(* Logix 5000 project; controller reports 1756-L63 rev 20.11; software revision 20.04; part 26 of 52 *)

        [1809].time.Day := 15, [1809].time.Hour := 23, [1809].time.Minute := 9, [1809].time.Second := 59, [1810].log_data[0].min := 1.0, [1810].log_data[0].max := 1.0, [1810].log_data[0].total := 300.0, [1810].log_data[0].time := 300.0, [1810].log_data[0].minminute := 10, [1810].log_data[0].maxminute := 10, [1810].log_data[0].valid := 1, [1810].log_data[1].valid := 1, [1810].log_data[2].valid := 1, [1810].log_data[3].valid := 1, [1810].log_data[4].valid := 1, [1810].log_data[5].valid := 1, [1810].log_data[6].valid := 1, [1810].log_data[7].valid := 1, [1810].log_data[8].valid := 1, [1810].log_data[9].valid := 1, [1810].log_data[10].valid := 1, [1810].log_data[11].valid := 1, [1810].log_data[12].valid := 1, [1810].log_data[13].valid := 1, [1810].log_data[14].valid := 1, [1810].log_data[15].valid := 1, [1810].log_data[16].valid := 1, [1810].log_data[17].valid := 1, [1810].log_data[18].valid := 1, [1810].log_data[19].valid := 1, [1810].time.Year := 2023, [1810].time.Month := 1, [1810].time.Day := 15, [1810].time.Hour := 23, [1810].time.Minute := 14, [1810].time.Second := 59, [1811].log_data[0].min := 1.0, [1811].log_data[0].max := 1.0, [1811].log_data[0].total := 300.0, [1811].log_data[0].time := 300.0, [1811].log_data[0].minminute := 15, [1811].log_data[0].maxminute := 15, [1811].log_data[0].valid := 1, [1811].log_data[1].valid := 1, [1811].log_data[2].valid := 1, [1811].log_data[3].valid := 1, [1811].log_data[4].valid := 1, [1811].log_data[5].valid := 1, [1811].log_data[6].valid := 1, [1811].log_data[7].valid := 1, [1811].log_data[8].valid := 1, [1811].log_data[9].valid := 1, [1811].log_data[10].valid := 1, [1811].log_data[11].valid := 1, [1811].log_data[12].valid := 1, [1811].log_data[13].valid := 1, [1811].log_data[14].valid := 1, [1811].log_data[15].valid := 1, [1811].log_data[16].valid := 1, [1811].log_data[17].valid := 1,
        [1811].log_data[18].valid := 1, [1811].log_data[19].valid := 1, [1811].time.Year := 2023, [1811].time.Month := 1, [1811].time.Day := 15, [1811].time.Hour := 23, [1811].time.Minute := 19, [1811].time.Second := 59, [1812].log_data[0].min := 1.0, [1812].log_data[0].max := 1.0, [1812].log_data[0].total := 300.0, [1812].log_data[0].time := 300.0, [1812].log_data[0].minminute := 20, [1812].log_data[0].maxminute := 20, [1812].log_data[0].valid := 1, [1812].log_data[1].valid := 1, [1812].log_data[2].valid := 1, [1812].log_data[3].valid := 1, [1812].log_data[4].valid := 1, [1812].log_data[5].valid := 1, [1812].log_data[6].valid := 1, [1812].log_data[7].valid := 1, [1812].log_data[8].valid := 1, [1812].log_data[9].valid := 1, [1812].log_data[10].valid := 1, [1812].log_data[11].valid := 1, [1812].log_data[12].valid := 1, [1812].log_data[13].valid := 1, [1812].log_data[14].valid := 1, [1812].log_data[15].valid := 1, [1812].log_data[16].valid := 1, [1812].log_data[17].valid := 1, [1812].log_data[18].valid := 1, [1812].log_data[19].valid := 1, [1812].time.Year := 2023, [1812].time.Month := 1, [1812].time.Day := 15, [1812].time.Hour := 23, [1812].time.Minute := 24, [1812].time.Second := 59, [1813].log_data[0].min := 1.0, [1813].log_data[0].max := 1.0, [1813].log_data[0].total := 300.0, [1813].log_data[0].time := 300.0, [1813].log_data[0].minminute := 25, [1813].log_data[0].maxminute := 25, [1813].log_data[0].valid := 1, [1813].log_data[1].valid := 1, [1813].log_data[2].valid := 1, [1813].log_data[3].valid := 1, [1813].log_data[4].valid := 1, [1813].log_data[5].valid := 1, [1813].log_data[6].valid := 1, [1813].log_data[7].valid := 1, [1813].log_data[8].valid := 1, [1813].log_data[9].valid := 1, [1813].log_data[10].valid := 1, [1813].log_data[11].valid := 1, [1813].log_data[12].valid := 1, [1813].log_data[13].valid := 1,
        [1813].log_data[14].valid := 1, [1813].log_data[15].valid := 1, [1813].log_data[16].valid := 1, [1813].log_data[17].valid := 1, [1813].log_data[18].valid := 1, [1813].log_data[19].valid := 1, [1813].time.Year := 2023, [1813].time.Month := 1, [1813].time.Day := 15, [1813].time.Hour := 23, [1813].time.Minute := 29, [1813].time.Second := 59, [1814].log_data[0].min := 1.0, [1814].log_data[0].max := 1.0, [1814].log_data[0].total := 300.0, [1814].log_data[0].time := 300.0, [1814].log_data[0].minminute := 30, [1814].log_data[0].maxminute := 30, [1814].log_data[0].valid := 1, [1814].log_data[1].valid := 1, [1814].log_data[2].valid := 1, [1814].log_data[3].valid := 1, [1814].log_data[4].valid := 1, [1814].log_data[5].valid := 1, [1814].log_data[6].valid := 1, [1814].log_data[7].valid := 1, [1814].log_data[8].valid := 1, [1814].log_data[9].valid := 1, [1814].log_data[10].valid := 1, [1814].log_data[11].valid := 1, [1814].log_data[12].valid := 1, [1814].log_data[13].valid := 1, [1814].log_data[14].valid := 1, [1814].log_data[15].valid := 1, [1814].log_data[16].valid := 1, [1814].log_data[17].valid := 1, [1814].log_data[18].valid := 1, [1814].log_data[19].valid := 1, [1814].time.Year := 2023, [1814].time.Month := 1, [1814].time.Day := 15, [1814].time.Hour := 23, [1814].time.Minute := 34, [1814].time.Second := 59, [1815].log_data[0].min := 1.0, [1815].log_data[0].max := 1.0, [1815].log_data[0].total := 300.0, [1815].log_data[0].time := 300.0, [1815].log_data[0].minminute := 35, [1815].log_data[0].maxminute := 35, [1815].log_data[0].valid := 1, [1815].log_data[1].valid := 1, [1815].log_data[2].valid := 1, [1815].log_data[3].valid := 1, [1815].log_data[4].valid := 1, [1815].log_data[5].valid := 1, [1815].log_data[6].valid := 1, [1815].log_data[7].valid := 1, [1815].log_data[8].valid := 1, [1815].log_data[9].valid := 1,
        [1815].log_data[10].valid := 1, [1815].log_data[11].valid := 1, [1815].log_data[12].valid := 1, [1815].log_data[13].valid := 1, [1815].log_data[14].valid := 1, [1815].log_data[15].valid := 1, [1815].log_data[16].valid := 1, [1815].log_data[17].valid := 1, [1815].log_data[18].valid := 1, [1815].log_data[19].valid := 1, [1815].time.Year := 2023, [1815].time.Month := 1, [1815].time.Day := 15, [1815].time.Hour := 23, [1815].time.Minute := 39, [1815].time.Second := 59, [1816].log_data[0].min := 1.0, [1816].log_data[0].max := 1.0, [1816].log_data[0].total := 300.0, [1816].log_data[0].time := 300.0, [1816].log_data[0].minminute := 40, [1816].log_data[0].maxminute := 40, [1816].log_data[0].valid := 1, [1816].log_data[1].valid := 1, [1816].log_data[2].valid := 1, [1816].log_data[3].valid := 1, [1816].log_data[4].valid := 1, [1816].log_data[5].valid := 1, [1816].log_data[6].valid := 1, [1816].log_data[7].valid := 1, [1816].log_data[8].valid := 1, [1816].log_data[9].valid := 1, [1816].log_data[10].valid := 1, [1816].log_data[11].valid := 1, [1816].log_data[12].valid := 1, [1816].log_data[13].valid := 1, [1816].log_data[14].valid := 1, [1816].log_data[15].valid := 1, [1816].log_data[16].valid := 1, [1816].log_data[17].valid := 1, [1816].log_data[18].valid := 1, [1816].log_data[19].valid := 1, [1816].time.Year := 2023, [1816].time.Month := 1, [1816].time.Day := 15, [1816].time.Hour := 23, [1816].time.Minute := 44, [1816].time.Second := 59, [1817].log_data[0].min := 1.0, [1817].log_data[0].max := 1.0, [1817].log_data[0].total := 300.0, [1817].log_data[0].time := 300.0, [1817].log_data[0].minminute := 45, [1817].log_data[0].maxminute := 45, [1817].log_data[0].valid := 1, [1817].log_data[1].valid := 1, [1817].log_data[2].valid := 1, [1817].log_data[3].valid := 1, [1817].log_data[4].valid := 1, [1817].log_data[5].valid := 1,
        [1817].log_data[6].valid := 1, [1817].log_data[7].valid := 1, [1817].log_data[8].valid := 1, [1817].log_data[9].valid := 1, [1817].log_data[10].valid := 1, [1817].log_data[11].valid := 1, [1817].log_data[12].valid := 1, [1817].log_data[13].valid := 1, [1817].log_data[14].valid := 1, [1817].log_data[15].valid := 1, [1817].log_data[16].valid := 1, [1817].log_data[17].valid := 1, [1817].log_data[18].valid := 1, [1817].log_data[19].valid := 1, [1817].time.Year := 2023, [1817].time.Month := 1, [1817].time.Day := 15, [1817].time.Hour := 23, [1817].time.Minute := 49, [1817].time.Second := 59, [1818].log_data[0].min := 1.0, [1818].log_data[0].max := 1.0, [1818].log_data[0].total := 300.0, [1818].log_data[0].time := 300.0, [1818].log_data[0].minminute := 50, [1818].log_data[0].maxminute := 50, [1818].log_data[0].valid := 1, [1818].log_data[1].valid := 1, [1818].log_data[2].valid := 1, [1818].log_data[3].valid := 1, [1818].log_data[4].valid := 1, [1818].log_data[5].valid := 1, [1818].log_data[6].valid := 1, [1818].log_data[7].valid := 1, [1818].log_data[8].valid := 1, [1818].log_data[9].valid := 1, [1818].log_data[10].valid := 1, [1818].log_data[11].valid := 1, [1818].log_data[12].valid := 1, [1818].log_data[13].valid := 1, [1818].log_data[14].valid := 1, [1818].log_data[15].valid := 1, [1818].log_data[16].valid := 1, [1818].log_data[17].valid := 1, [1818].log_data[18].valid := 1, [1818].log_data[19].valid := 1, [1818].time.Year := 2023, [1818].time.Month := 1, [1818].time.Day := 15, [1818].time.Hour := 23, [1818].time.Minute := 54, [1818].time.Second := 59, [1819].log_data[0].min := 1.0, [1819].log_data[0].max := 1.0, [1819].log_data[0].total := 300.0, [1819].log_data[0].time := 300.0, [1819].log_data[0].minminute := 55, [1819].log_data[0].maxminute := 55, [1819].log_data[0].valid := 1, [1819].log_data[1].valid := 1,
        [1819].log_data[2].valid := 1, [1819].log_data[3].valid := 1, [1819].log_data[4].valid := 1, [1819].log_data[5].valid := 1, [1819].log_data[6].valid := 1, [1819].log_data[7].valid := 1, [1819].log_data[8].valid := 1, [1819].log_data[9].valid := 1, [1819].log_data[10].valid := 1, [1819].log_data[11].valid := 1, [1819].log_data[12].valid := 1, [1819].log_data[13].valid := 1, [1819].log_data[14].valid := 1, [1819].log_data[15].valid := 1, [1819].log_data[16].valid := 1, [1819].log_data[17].valid := 1, [1819].log_data[18].valid := 1, [1819].log_data[19].valid := 1, [1819].time.Year := 2023, [1819].time.Month := 1, [1819].time.Day := 15, [1819].time.Hour := 23, [1819].time.Minute := 59, [1819].time.Second := 59, [1820].log_data[0].min := 1.0, [1820].log_data[0].max := 1.0, [1820].log_data[0].total := 300.0, [1820].log_data[0].time := 300.0, [1820].log_data[0].valid := 1, [1820].log_data[1].valid := 1, [1820].log_data[2].valid := 1, [1820].log_data[3].valid := 1, [1820].log_data[4].valid := 1, [1820].log_data[5].valid := 1, [1820].log_data[6].valid := 1, [1820].log_data[7].valid := 1, [1820].log_data[8].valid := 1, [1820].log_data[9].valid := 1, [1820].log_data[10].valid := 1, [1820].log_data[11].valid := 1, [1820].log_data[12].valid := 1, [1820].log_data[13].valid := 1, [1820].log_data[14].valid := 1, [1820].log_data[15].valid := 1, [1820].log_data[16].valid := 1, [1820].log_data[17].valid := 1, [1820].log_data[18].valid := 1, [1820].log_data[19].valid := 1, [1820].time.Year := 2023, [1820].time.Month := 1, [1820].time.Day := 16, [1820].time.Minute := 4, [1820].time.Second := 59, [1821].log_data[0].min := 1.0, [1821].log_data[0].max := 1.0, [1821].log_data[0].total := 300.0, [1821].log_data[0].time := 300.0, [1821].log_data[0].minminute := 5, [1821].log_data[0].maxminute := 5, [1821].log_data[0].valid := 1,
        [1821].log_data[1].valid := 1, [1821].log_data[2].valid := 1, [1821].log_data[3].valid := 1, [1821].log_data[4].valid := 1, [1821].log_data[5].valid := 1, [1821].log_data[6].valid := 1, [1821].log_data[7].valid := 1, [1821].log_data[8].valid := 1, [1821].log_data[9].valid := 1, [1821].log_data[10].valid := 1, [1821].log_data[11].valid := 1, [1821].log_data[12].valid := 1, [1821].log_data[13].valid := 1, [1821].log_data[14].valid := 1, [1821].log_data[15].valid := 1, [1821].log_data[16].valid := 1, [1821].log_data[17].valid := 1, [1821].log_data[18].valid := 1, [1821].log_data[19].valid := 1, [1821].time.Year := 2023, [1821].time.Month := 1, [1821].time.Day := 16, [1821].time.Minute := 9, [1821].time.Second := 59, [1822].log_data[0].min := 1.0, [1822].log_data[0].max := 1.0, [1822].log_data[0].total := 300.0, [1822].log_data[0].time := 300.0, [1822].log_data[0].minminute := 10, [1822].log_data[0].maxminute := 10, [1822].log_data[0].valid := 1, [1822].log_data[1].valid := 1, [1822].log_data[2].valid := 1, [1822].log_data[3].valid := 1, [1822].log_data[4].valid := 1, [1822].log_data[5].valid := 1, [1822].log_data[6].valid := 1, [1822].log_data[7].valid := 1, [1822].log_data[8].valid := 1, [1822].log_data[9].valid := 1, [1822].log_data[10].valid := 1, [1822].log_data[11].valid := 1, [1822].log_data[12].valid := 1, [1822].log_data[13].valid := 1, [1822].log_data[14].valid := 1, [1822].log_data[15].valid := 1, [1822].log_data[16].valid := 1, [1822].log_data[17].valid := 1, [1822].log_data[18].valid := 1, [1822].log_data[19].valid := 1, [1822].time.Year := 2023, [1822].time.Month := 1, [1822].time.Day := 16, [1822].time.Minute := 14, [1822].time.Second := 59, [1823].log_data[0].min := 1.0, [1823].log_data[0].max := 1.0, [1823].log_data[0].total := 300.0, [1823].log_data[0].time := 300.0, [1823].log_data[0].minminute := 15,
        [1823].log_data[0].maxminute := 15, [1823].log_data[0].valid := 1, [1823].log_data[1].valid := 1, [1823].log_data[2].valid := 1, [1823].log_data[3].valid := 1, [1823].log_data[4].valid := 1, [1823].log_data[5].valid := 1, [1823].log_data[6].valid := 1, [1823].log_data[7].valid := 1, [1823].log_data[8].valid := 1, [1823].log_data[9].valid := 1, [1823].log_data[10].valid := 1, [1823].log_data[11].valid := 1, [1823].log_data[12].valid := 1, [1823].log_data[13].valid := 1, [1823].log_data[14].valid := 1, [1823].log_data[15].valid := 1, [1823].log_data[16].valid := 1, [1823].log_data[17].valid := 1, [1823].log_data[18].valid := 1, [1823].log_data[19].valid := 1, [1823].time.Year := 2023, [1823].time.Month := 1, [1823].time.Day := 16, [1823].time.Minute := 19, [1823].time.Second := 59, [1824].log_data[0].min := 1.0, [1824].log_data[0].max := 1.0, [1824].log_data[0].total := 300.0, [1824].log_data[0].time := 300.0, [1824].log_data[0].minminute := 20, [1824].log_data[0].maxminute := 20, [1824].log_data[0].valid := 1, [1824].log_data[1].valid := 1, [1824].log_data[2].valid := 1, [1824].log_data[3].valid := 1, [1824].log_data[4].valid := 1, [1824].log_data[5].valid := 1, [1824].log_data[6].valid := 1, [1824].log_data[7].valid := 1, [1824].log_data[8].valid := 1, [1824].log_data[9].valid := 1, [1824].log_data[10].valid := 1, [1824].log_data[11].valid := 1, [1824].log_data[12].valid := 1, [1824].log_data[13].valid := 1, [1824].log_data[14].valid := 1, [1824].log_data[15].valid := 1, [1824].log_data[16].valid := 1, [1824].log_data[17].valid := 1, [1824].log_data[18].valid := 1, [1824].log_data[19].valid := 1, [1824].time.Year := 2023, [1824].time.Month := 1, [1824].time.Day := 16, [1824].time.Minute := 24, [1824].time.Second := 59, [1825].log_data[0].min := 1.0, [1825].log_data[0].max := 1.0, [1825].log_data[0].total := 300.0,
        [1825].log_data[0].time := 300.0, [1825].log_data[0].minminute := 25, [1825].log_data[0].maxminute := 25, [1825].log_data[0].valid := 1, [1825].log_data[1].valid := 1, [1825].log_data[2].valid := 1, [1825].log_data[3].valid := 1, [1825].log_data[4].valid := 1, [1825].log_data[5].valid := 1, [1825].log_data[6].valid := 1, [1825].log_data[7].valid := 1, [1825].log_data[8].valid := 1, [1825].log_data[9].valid := 1, [1825].log_data[10].valid := 1, [1825].log_data[11].valid := 1, [1825].log_data[12].valid := 1, [1825].log_data[13].valid := 1, [1825].log_data[14].valid := 1, [1825].log_data[15].valid := 1, [1825].log_data[16].valid := 1, [1825].log_data[17].valid := 1, [1825].log_data[18].valid := 1, [1825].log_data[19].valid := 1, [1825].time.Year := 2023, [1825].time.Month := 1, [1825].time.Day := 16, [1825].time.Minute := 29, [1825].time.Second := 59, [1826].log_data[0].min := 1.0, [1826].log_data[0].max := 1.0, [1826].log_data[0].total := 300.0, [1826].log_data[0].time := 300.0, [1826].log_data[0].minminute := 30, [1826].log_data[0].maxminute := 30, [1826].log_data[0].valid := 1, [1826].log_data[1].valid := 1, [1826].log_data[2].valid := 1, [1826].log_data[3].valid := 1, [1826].log_data[4].valid := 1, [1826].log_data[5].valid := 1, [1826].log_data[6].valid := 1, [1826].log_data[7].valid := 1, [1826].log_data[8].valid := 1, [1826].log_data[9].valid := 1, [1826].log_data[10].valid := 1, [1826].log_data[11].valid := 1, [1826].log_data[12].valid := 1, [1826].log_data[13].valid := 1, [1826].log_data[14].valid := 1, [1826].log_data[15].valid := 1, [1826].log_data[16].valid := 1, [1826].log_data[17].valid := 1, [1826].log_data[18].valid := 1, [1826].log_data[19].valid := 1, [1826].time.Year := 2023, [1826].time.Month := 1, [1826].time.Day := 16, [1826].time.Minute := 34, [1826].time.Second := 59, [1827].log_data[0].min := 1.0,
        [1827].log_data[0].max := 1.0, [1827].log_data[0].total := 300.0, [1827].log_data[0].time := 300.0, [1827].log_data[0].minminute := 35, [1827].log_data[0].maxminute := 35, [1827].log_data[0].valid := 1, [1827].log_data[1].valid := 1, [1827].log_data[2].valid := 1, [1827].log_data[3].valid := 1, [1827].log_data[4].valid := 1, [1827].log_data[5].valid := 1, [1827].log_data[6].valid := 1, [1827].log_data[7].valid := 1, [1827].log_data[8].valid := 1, [1827].log_data[9].valid := 1, [1827].log_data[10].valid := 1, [1827].log_data[11].valid := 1, [1827].log_data[12].valid := 1, [1827].log_data[13].valid := 1, [1827].log_data[14].valid := 1, [1827].log_data[15].valid := 1, [1827].log_data[16].valid := 1, [1827].log_data[17].valid := 1, [1827].log_data[18].valid := 1, [1827].log_data[19].valid := 1, [1827].time.Year := 2023, [1827].time.Month := 1, [1827].time.Day := 16, [1827].time.Minute := 39, [1827].time.Second := 59, [1828].log_data[0].min := 1.0, [1828].log_data[0].max := 1.0, [1828].log_data[0].total := 300.0, [1828].log_data[0].time := 300.0, [1828].log_data[0].minminute := 40, [1828].log_data[0].maxminute := 40, [1828].log_data[0].valid := 1, [1828].log_data[1].valid := 1, [1828].log_data[2].valid := 1, [1828].log_data[3].valid := 1, [1828].log_data[4].valid := 1, [1828].log_data[5].valid := 1, [1828].log_data[6].valid := 1, [1828].log_data[7].valid := 1, [1828].log_data[8].valid := 1, [1828].log_data[9].valid := 1, [1828].log_data[10].valid := 1, [1828].log_data[11].valid := 1, [1828].log_data[12].valid := 1, [1828].log_data[13].valid := 1, [1828].log_data[14].valid := 1, [1828].log_data[15].valid := 1, [1828].log_data[16].valid := 1, [1828].log_data[17].valid := 1, [1828].log_data[18].valid := 1, [1828].log_data[19].valid := 1, [1828].time.Year := 2023, [1828].time.Month := 1, [1828].time.Day := 16, [1828].time.Minute := 44,
        [1828].time.Second := 59, [1829].log_data[0].min := 1.0, [1829].log_data[0].max := 1.0, [1829].log_data[0].total := 300.0, [1829].log_data[0].time := 300.0, [1829].log_data[0].minminute := 45, [1829].log_data[0].maxminute := 45, [1829].log_data[0].valid := 1, [1829].log_data[1].valid := 1, [1829].log_data[2].valid := 1, [1829].log_data[3].valid := 1, [1829].log_data[4].valid := 1, [1829].log_data[5].valid := 1, [1829].log_data[6].valid := 1, [1829].log_data[7].valid := 1, [1829].log_data[8].valid := 1, [1829].log_data[9].valid := 1, [1829].log_data[10].valid := 1, [1829].log_data[11].valid := 1, [1829].log_data[12].valid := 1, [1829].log_data[13].valid := 1, [1829].log_data[14].valid := 1, [1829].log_data[15].valid := 1, [1829].log_data[16].valid := 1, [1829].log_data[17].valid := 1, [1829].log_data[18].valid := 1, [1829].log_data[19].valid := 1, [1829].time.Year := 2023, [1829].time.Month := 1, [1829].time.Day := 16, [1829].time.Minute := 49, [1829].time.Second := 59, [1830].log_data[0].min := 1.0, [1830].log_data[0].max := 1.0, [1830].log_data[0].total := 300.0, [1830].log_data[0].time := 300.0, [1830].log_data[0].minminute := 50, [1830].log_data[0].maxminute := 50, [1830].log_data[0].valid := 1, [1830].log_data[1].valid := 1, [1830].log_data[2].valid := 1, [1830].log_data[3].valid := 1, [1830].log_data[4].valid := 1, [1830].log_data[5].valid := 1, [1830].log_data[6].valid := 1, [1830].log_data[7].valid := 1, [1830].log_data[8].valid := 1, [1830].log_data[9].valid := 1, [1830].log_data[10].valid := 1, [1830].log_data[11].valid := 1, [1830].log_data[12].valid := 1, [1830].log_data[13].valid := 1, [1830].log_data[14].valid := 1, [1830].log_data[15].valid := 1, [1830].log_data[16].valid := 1, [1830].log_data[17].valid := 1, [1830].log_data[18].valid := 1, [1830].log_data[19].valid := 1, [1830].time.Year := 2023, [1830].time.Month := 1,
        [1830].time.Day := 16, [1830].time.Minute := 54, [1830].time.Second := 59, [1831].log_data[0].min := 1.0, [1831].log_data[0].max := 1.0, [1831].log_data[0].total := 300.0, [1831].log_data[0].time := 300.0, [1831].log_data[0].minminute := 55, [1831].log_data[0].maxminute := 55, [1831].log_data[0].valid := 1, [1831].log_data[1].valid := 1, [1831].log_data[2].valid := 1, [1831].log_data[3].valid := 1, [1831].log_data[4].valid := 1, [1831].log_data[5].valid := 1, [1831].log_data[6].valid := 1, [1831].log_data[7].valid := 1, [1831].log_data[8].valid := 1, [1831].log_data[9].valid := 1, [1831].log_data[10].valid := 1, [1831].log_data[11].valid := 1, [1831].log_data[12].valid := 1, [1831].log_data[13].valid := 1, [1831].log_data[14].valid := 1, [1831].log_data[15].valid := 1, [1831].log_data[16].valid := 1, [1831].log_data[17].valid := 1, [1831].log_data[18].valid := 1, [1831].log_data[19].valid := 1, [1831].time.Year := 2023, [1831].time.Month := 1, [1831].time.Day := 16, [1831].time.Minute := 59, [1831].time.Second := 59, [1832].log_data[0].min := 1.0, [1832].log_data[0].max := 1.0, [1832].log_data[0].total := 300.0, [1832].log_data[0].time := 300.0, [1832].log_data[0].valid := 1, [1832].log_data[1].valid := 1, [1832].log_data[2].valid := 1, [1832].log_data[3].valid := 1, [1832].log_data[4].valid := 1, [1832].log_data[5].valid := 1, [1832].log_data[6].valid := 1, [1832].log_data[7].valid := 1, [1832].log_data[8].valid := 1, [1832].log_data[9].valid := 1, [1832].log_data[10].valid := 1, [1832].log_data[11].valid := 1, [1832].log_data[12].valid := 1, [1832].log_data[13].valid := 1, [1832].log_data[14].valid := 1, [1832].log_data[15].valid := 1, [1832].log_data[16].valid := 1, [1832].log_data[17].valid := 1, [1832].log_data[18].valid := 1, [1832].log_data[19].valid := 1, [1832].time.Year := 2023, [1832].time.Month := 1,
        [1832].time.Day := 16, [1832].time.Hour := 1, [1832].time.Minute := 4, [1832].time.Second := 59, [1833].log_data[0].min := 1.0, [1833].log_data[0].max := 1.0, [1833].log_data[0].total := 300.0, [1833].log_data[0].time := 300.0, [1833].log_data[0].minminute := 5, [1833].log_data[0].maxminute := 5, [1833].log_data[0].valid := 1, [1833].log_data[1].valid := 1, [1833].log_data[2].valid := 1, [1833].log_data[3].valid := 1, [1833].log_data[4].valid := 1, [1833].log_data[5].valid := 1, [1833].log_data[6].valid := 1, [1833].log_data[7].valid := 1, [1833].log_data[8].valid := 1, [1833].log_data[9].valid := 1, [1833].log_data[10].valid := 1, [1833].log_data[11].valid := 1, [1833].log_data[12].valid := 1, [1833].log_data[13].valid := 1, [1833].log_data[14].valid := 1, [1833].log_data[15].valid := 1, [1833].log_data[16].valid := 1, [1833].log_data[17].valid := 1, [1833].log_data[18].valid := 1, [1833].log_data[19].valid := 1, [1833].time.Year := 2023, [1833].time.Month := 1, [1833].time.Day := 16, [1833].time.Hour := 1, [1833].time.Minute := 9, [1833].time.Second := 59, [1834].log_data[0].min := 1.0, [1834].log_data[0].max := 1.0, [1834].log_data[0].total := 300.0, [1834].log_data[0].time := 300.0, [1834].log_data[0].minminute := 10, [1834].log_data[0].maxminute := 10, [1834].log_data[0].valid := 1, [1834].log_data[1].valid := 1, [1834].log_data[2].valid := 1, [1834].log_data[3].valid := 1, [1834].log_data[4].valid := 1, [1834].log_data[5].valid := 1, [1834].log_data[6].valid := 1, [1834].log_data[7].valid := 1, [1834].log_data[8].valid := 1, [1834].log_data[9].valid := 1, [1834].log_data[10].valid := 1, [1834].log_data[11].valid := 1, [1834].log_data[12].valid := 1, [1834].log_data[13].valid := 1, [1834].log_data[14].valid := 1, [1834].log_data[15].valid := 1, [1834].log_data[16].valid := 1, [1834].log_data[17].valid := 1,
        [1834].log_data[18].valid := 1, [1834].log_data[19].valid := 1, [1834].time.Year := 2023, [1834].time.Month := 1, [1834].time.Day := 16, [1834].time.Hour := 1, [1834].time.Minute := 14, [1834].time.Second := 59, [1835].log_data[0].min := 1.0, [1835].log_data[0].max := 1.0, [1835].log_data[0].total := 300.0, [1835].log_data[0].time := 300.0, [1835].log_data[0].minminute := 15, [1835].log_data[0].maxminute := 15, [1835].log_data[0].valid := 1, [1835].log_data[1].valid := 1, [1835].log_data[2].valid := 1, [1835].log_data[3].valid := 1, [1835].log_data[4].valid := 1, [1835].log_data[5].valid := 1, [1835].log_data[6].valid := 1, [1835].log_data[7].valid := 1, [1835].log_data[8].valid := 1, [1835].log_data[9].valid := 1, [1835].log_data[10].valid := 1, [1835].log_data[11].valid := 1, [1835].log_data[12].valid := 1, [1835].log_data[13].valid := 1, [1835].log_data[14].valid := 1, [1835].log_data[15].valid := 1, [1835].log_data[16].valid := 1, [1835].log_data[17].valid := 1, [1835].log_data[18].valid := 1, [1835].log_data[19].valid := 1, [1835].time.Year := 2023, [1835].time.Month := 1, [1835].time.Day := 16, [1835].time.Hour := 1, [1835].time.Minute := 19, [1835].time.Second := 59, [1836].log_data[0].min := 1.0, [1836].log_data[0].max := 1.0, [1836].log_data[0].total := 300.0, [1836].log_data[0].time := 300.0, [1836].log_data[0].minminute := 20, [1836].log_data[0].maxminute := 20, [1836].log_data[0].valid := 1, [1836].log_data[1].valid := 1, [1836].log_data[2].valid := 1, [1836].log_data[3].valid := 1, [1836].log_data[4].valid := 1, [1836].log_data[5].valid := 1, [1836].log_data[6].valid := 1, [1836].log_data[7].valid := 1, [1836].log_data[8].valid := 1, [1836].log_data[9].valid := 1, [1836].log_data[10].valid := 1, [1836].log_data[11].valid := 1, [1836].log_data[12].valid := 1, [1836].log_data[13].valid := 1,
        [1836].log_data[14].valid := 1, [1836].log_data[15].valid := 1, [1836].log_data[16].valid := 1, [1836].log_data[17].valid := 1, [1836].log_data[18].valid := 1, [1836].log_data[19].valid := 1, [1836].time.Year := 2023, [1836].time.Month := 1, [1836].time.Day := 16, [1836].time.Hour := 1, [1836].time.Minute := 24, [1836].time.Second := 59, [1837].log_data[0].min := 1.0, [1837].log_data[0].max := 1.0, [1837].log_data[0].total := 300.0, [1837].log_data[0].time := 300.0, [1837].log_data[0].minminute := 25, [1837].log_data[0].maxminute := 25, [1837].log_data[0].valid := 1, [1837].log_data[1].valid := 1, [1837].log_data[2].valid := 1, [1837].log_data[3].valid := 1, [1837].log_data[4].valid := 1, [1837].log_data[5].valid := 1, [1837].log_data[6].valid := 1, [1837].log_data[7].valid := 1, [1837].log_data[8].valid := 1, [1837].log_data[9].valid := 1, [1837].log_data[10].valid := 1, [1837].log_data[11].valid := 1, [1837].log_data[12].valid := 1, [1837].log_data[13].valid := 1, [1837].log_data[14].valid := 1, [1837].log_data[15].valid := 1, [1837].log_data[16].valid := 1, [1837].log_data[17].valid := 1, [1837].log_data[18].valid := 1, [1837].log_data[19].valid := 1, [1837].time.Year := 2023, [1837].time.Month := 1, [1837].time.Day := 16, [1837].time.Hour := 1, [1837].time.Minute := 29, [1837].time.Second := 59, [1838].log_data[0].min := 1.0, [1838].log_data[0].max := 1.0, [1838].log_data[0].total := 300.0, [1838].log_data[0].time := 300.0, [1838].log_data[0].minminute := 30, [1838].log_data[0].maxminute := 30, [1838].log_data[0].valid := 1, [1838].log_data[1].valid := 1, [1838].log_data[2].valid := 1, [1838].log_data[3].valid := 1, [1838].log_data[4].valid := 1, [1838].log_data[5].valid := 1, [1838].log_data[6].valid := 1, [1838].log_data[7].valid := 1, [1838].log_data[8].valid := 1, [1838].log_data[9].valid := 1,
        [1838].log_data[10].valid := 1, [1838].log_data[11].valid := 1, [1838].log_data[12].valid := 1, [1838].log_data[13].valid := 1, [1838].log_data[14].valid := 1, [1838].log_data[15].valid := 1, [1838].log_data[16].valid := 1, [1838].log_data[17].valid := 1, [1838].log_data[18].valid := 1, [1838].log_data[19].valid := 1, [1838].time.Year := 2023, [1838].time.Month := 1, [1838].time.Day := 16, [1838].time.Hour := 1, [1838].time.Minute := 34, [1838].time.Second := 59, [1839].log_data[0].min := 1.0, [1839].log_data[0].max := 1.0, [1839].log_data[0].total := 300.0, [1839].log_data[0].time := 300.0, [1839].log_data[0].minminute := 35, [1839].log_data[0].maxminute := 35, [1839].log_data[0].valid := 1, [1839].log_data[1].valid := 1, [1839].log_data[2].valid := 1, [1839].log_data[3].valid := 1, [1839].log_data[4].valid := 1, [1839].log_data[5].valid := 1, [1839].log_data[6].valid := 1, [1839].log_data[7].valid := 1, [1839].log_data[8].valid := 1, [1839].log_data[9].valid := 1, [1839].log_data[10].valid := 1, [1839].log_data[11].valid := 1, [1839].log_data[12].valid := 1, [1839].log_data[13].valid := 1, [1839].log_data[14].valid := 1, [1839].log_data[15].valid := 1, [1839].log_data[16].valid := 1, [1839].log_data[17].valid := 1, [1839].log_data[18].valid := 1, [1839].log_data[19].valid := 1, [1839].time.Year := 2023, [1839].time.Month := 1, [1839].time.Day := 16, [1839].time.Hour := 1, [1839].time.Minute := 39, [1839].time.Second := 59, [1840].log_data[0].min := 1.0, [1840].log_data[0].max := 1.0, [1840].log_data[0].total := 300.0, [1840].log_data[0].time := 300.0, [1840].log_data[0].minminute := 40, [1840].log_data[0].maxminute := 40, [1840].log_data[0].valid := 1, [1840].log_data[1].valid := 1, [1840].log_data[2].valid := 1, [1840].log_data[3].valid := 1, [1840].log_data[4].valid := 1, [1840].log_data[5].valid := 1,
        [1840].log_data[6].valid := 1, [1840].log_data[7].valid := 1, [1840].log_data[8].valid := 1, [1840].log_data[9].valid := 1, [1840].log_data[10].valid := 1, [1840].log_data[11].valid := 1, [1840].log_data[12].valid := 1, [1840].log_data[13].valid := 1, [1840].log_data[14].valid := 1, [1840].log_data[15].valid := 1, [1840].log_data[16].valid := 1, [1840].log_data[17].valid := 1, [1840].log_data[18].valid := 1, [1840].log_data[19].valid := 1, [1840].time.Year := 2023, [1840].time.Month := 1, [1840].time.Day := 16, [1840].time.Hour := 1, [1840].time.Minute := 44, [1840].time.Second := 59, [1841].log_data[0].min := 1.0, [1841].log_data[0].max := 1.0, [1841].log_data[0].total := 300.0, [1841].log_data[0].time := 300.0, [1841].log_data[0].minminute := 45, [1841].log_data[0].maxminute := 45, [1841].log_data[0].valid := 1, [1841].log_data[1].valid := 1, [1841].log_data[2].valid := 1, [1841].log_data[3].valid := 1, [1841].log_data[4].valid := 1, [1841].log_data[5].valid := 1, [1841].log_data[6].valid := 1, [1841].log_data[7].valid := 1, [1841].log_data[8].valid := 1, [1841].log_data[9].valid := 1, [1841].log_data[10].valid := 1, [1841].log_data[11].valid := 1, [1841].log_data[12].valid := 1, [1841].log_data[13].valid := 1, [1841].log_data[14].valid := 1, [1841].log_data[15].valid := 1, [1841].log_data[16].valid := 1, [1841].log_data[17].valid := 1, [1841].log_data[18].valid := 1, [1841].log_data[19].valid := 1, [1841].time.Year := 2023, [1841].time.Month := 1, [1841].time.Day := 16, [1841].time.Hour := 1, [1841].time.Minute := 49, [1841].time.Second := 59, [1842].log_data[0].min := 1.0, [1842].log_data[0].max := 1.0, [1842].log_data[0].total := 300.0, [1842].log_data[0].time := 300.0, [1842].log_data[0].minminute := 50, [1842].log_data[0].maxminute := 50, [1842].log_data[0].valid := 1, [1842].log_data[1].valid := 1,
        [1842].log_data[2].valid := 1, [1842].log_data[3].valid := 1, [1842].log_data[4].valid := 1, [1842].log_data[5].valid := 1, [1842].log_data[6].valid := 1, [1842].log_data[7].valid := 1, [1842].log_data[8].valid := 1, [1842].log_data[9].valid := 1, [1842].log_data[10].valid := 1, [1842].log_data[11].valid := 1, [1842].log_data[12].valid := 1, [1842].log_data[13].valid := 1, [1842].log_data[14].valid := 1, [1842].log_data[15].valid := 1, [1842].log_data[16].valid := 1, [1842].log_data[17].valid := 1, [1842].log_data[18].valid := 1, [1842].log_data[19].valid := 1, [1842].time.Year := 2023, [1842].time.Month := 1, [1842].time.Day := 16, [1842].time.Hour := 1, [1842].time.Minute := 54, [1842].time.Second := 59, [1843].log_data[0].min := 1.0, [1843].log_data[0].max := 1.0, [1843].log_data[0].total := 300.0, [1843].log_data[0].time := 300.0, [1843].log_data[0].minminute := 55, [1843].log_data[0].maxminute := 55, [1843].log_data[0].valid := 1, [1843].log_data[1].valid := 1, [1843].log_data[2].valid := 1, [1843].log_data[3].valid := 1, [1843].log_data[4].valid := 1, [1843].log_data[5].valid := 1, [1843].log_data[6].valid := 1, [1843].log_data[7].valid := 1, [1843].log_data[8].valid := 1, [1843].log_data[9].valid := 1, [1843].log_data[10].valid := 1, [1843].log_data[11].valid := 1, [1843].log_data[12].valid := 1, [1843].log_data[13].valid := 1, [1843].log_data[14].valid := 1, [1843].log_data[15].valid := 1, [1843].log_data[16].valid := 1, [1843].log_data[17].valid := 1, [1843].log_data[18].valid := 1, [1843].log_data[19].valid := 1, [1843].time.Year := 2023, [1843].time.Month := 1, [1843].time.Day := 16, [1843].time.Hour := 1, [1843].time.Minute := 59, [1843].time.Second := 59, [1844].log_data[0].min := 1.0, [1844].log_data[0].max := 1.0, [1844].log_data[0].total := 300.0, [1844].log_data[0].time := 300.0,
        [1844].log_data[0].valid := 1, [1844].log_data[1].valid := 1, [1844].log_data[2].valid := 1, [1844].log_data[3].valid := 1, [1844].log_data[4].valid := 1, [1844].log_data[5].valid := 1, [1844].log_data[6].valid := 1, [1844].log_data[7].valid := 1, [1844].log_data[8].valid := 1, [1844].log_data[9].valid := 1, [1844].log_data[10].valid := 1, [1844].log_data[11].valid := 1, [1844].log_data[12].valid := 1, [1844].log_data[13].valid := 1, [1844].log_data[14].valid := 1, [1844].log_data[15].valid := 1, [1844].log_data[16].valid := 1, [1844].log_data[17].valid := 1, [1844].log_data[18].valid := 1, [1844].log_data[19].valid := 1, [1844].time.Year := 2023, [1844].time.Month := 1, [1844].time.Day := 16, [1844].time.Hour := 2, [1844].time.Minute := 4, [1844].time.Second := 59, [1845].log_data[0].min := 1.0, [1845].log_data[0].max := 1.0, [1845].log_data[0].total := 300.0, [1845].log_data[0].time := 300.0, [1845].log_data[0].minminute := 5, [1845].log_data[0].maxminute := 5, [1845].log_data[0].valid := 1, [1845].log_data[1].valid := 1, [1845].log_data[2].valid := 1, [1845].log_data[3].valid := 1, [1845].log_data[4].valid := 1, [1845].log_data[5].valid := 1, [1845].log_data[6].valid := 1, [1845].log_data[7].valid := 1, [1845].log_data[8].valid := 1, [1845].log_data[9].valid := 1, [1845].log_data[10].valid := 1, [1845].log_data[11].valid := 1, [1845].log_data[12].valid := 1, [1845].log_data[13].valid := 1, [1845].log_data[14].valid := 1, [1845].log_data[15].valid := 1, [1845].log_data[16].valid := 1, [1845].log_data[17].valid := 1, [1845].log_data[18].valid := 1, [1845].log_data[19].valid := 1, [1845].time.Year := 2023, [1845].time.Month := 1, [1845].time.Day := 16, [1845].time.Hour := 2, [1845].time.Minute := 9, [1845].time.Second := 59, [1846].log_data[0].min := 1.0, [1846].log_data[0].max := 1.0,
        [1846].log_data[0].total := 300.0, [1846].log_data[0].time := 300.0, [1846].log_data[0].minminute := 10, [1846].log_data[0].maxminute := 10, [1846].log_data[0].valid := 1, [1846].log_data[1].valid := 1, [1846].log_data[2].valid := 1, [1846].log_data[3].valid := 1, [1846].log_data[4].valid := 1, [1846].log_data[5].valid := 1, [1846].log_data[6].valid := 1, [1846].log_data[7].valid := 1, [1846].log_data[8].valid := 1, [1846].log_data[9].valid := 1, [1846].log_data[10].valid := 1, [1846].log_data[11].valid := 1, [1846].log_data[12].valid := 1, [1846].log_data[13].valid := 1, [1846].log_data[14].valid := 1, [1846].log_data[15].valid := 1, [1846].log_data[16].valid := 1, [1846].log_data[17].valid := 1, [1846].log_data[18].valid := 1, [1846].log_data[19].valid := 1, [1846].time.Year := 2023, [1846].time.Month := 1, [1846].time.Day := 16, [1846].time.Hour := 2, [1846].time.Minute := 14, [1846].time.Second := 59, [1847].log_data[0].min := 1.0, [1847].log_data[0].max := 1.0, [1847].log_data[0].total := 300.0, [1847].log_data[0].time := 300.0, [1847].log_data[0].minminute := 15, [1847].log_data[0].maxminute := 15, [1847].log_data[0].valid := 1, [1847].log_data[1].valid := 1, [1847].log_data[2].valid := 1, [1847].log_data[3].valid := 1, [1847].log_data[4].valid := 1, [1847].log_data[5].valid := 1, [1847].log_data[6].valid := 1, [1847].log_data[7].valid := 1, [1847].log_data[8].valid := 1, [1847].log_data[9].valid := 1, [1847].log_data[10].valid := 1, [1847].log_data[11].valid := 1, [1847].log_data[12].valid := 1, [1847].log_data[13].valid := 1, [1847].log_data[14].valid := 1, [1847].log_data[15].valid := 1, [1847].log_data[16].valid := 1, [1847].log_data[17].valid := 1, [1847].log_data[18].valid := 1, [1847].log_data[19].valid := 1, [1847].time.Year := 2023, [1847].time.Month := 1, [1847].time.Day := 16, [1847].time.Hour := 2,
        [1847].time.Minute := 19, [1847].time.Second := 59, [1848].log_data[0].min := 1.0, [1848].log_data[0].max := 1.0, [1848].log_data[0].total := 300.0, [1848].log_data[0].time := 300.0, [1848].log_data[0].minminute := 20, [1848].log_data[0].maxminute := 20, [1848].log_data[0].valid := 1, [1848].log_data[1].valid := 1, [1848].log_data[2].valid := 1, [1848].log_data[3].valid := 1, [1848].log_data[4].valid := 1, [1848].log_data[5].valid := 1, [1848].log_data[6].valid := 1, [1848].log_data[7].valid := 1, [1848].log_data[8].valid := 1, [1848].log_data[9].valid := 1, [1848].log_data[10].valid := 1, [1848].log_data[11].valid := 1, [1848].log_data[12].valid := 1, [1848].log_data[13].valid := 1, [1848].log_data[14].valid := 1, [1848].log_data[15].valid := 1, [1848].log_data[16].valid := 1, [1848].log_data[17].valid := 1, [1848].log_data[18].valid := 1, [1848].log_data[19].valid := 1, [1848].time.Year := 2023, [1848].time.Month := 1, [1848].time.Day := 16, [1848].time.Hour := 2, [1848].time.Minute := 24, [1848].time.Second := 59, [1849].log_data[0].min := 1.0, [1849].log_data[0].max := 1.0, [1849].log_data[0].total := 300.0, [1849].log_data[0].time := 300.0, [1849].log_data[0].minminute := 25, [1849].log_data[0].maxminute := 25, [1849].log_data[0].valid := 1, [1849].log_data[1].valid := 1, [1849].log_data[2].valid := 1, [1849].log_data[3].valid := 1, [1849].log_data[4].valid := 1, [1849].log_data[5].valid := 1, [1849].log_data[6].valid := 1, [1849].log_data[7].valid := 1, [1849].log_data[8].valid := 1, [1849].log_data[9].valid := 1, [1849].log_data[10].valid := 1, [1849].log_data[11].valid := 1, [1849].log_data[12].valid := 1, [1849].log_data[13].valid := 1, [1849].log_data[14].valid := 1, [1849].log_data[15].valid := 1, [1849].log_data[16].valid := 1, [1849].log_data[17].valid := 1, [1849].log_data[18].valid := 1, [1849].log_data[19].valid := 1,
        [1849].time.Year := 2023, [1849].time.Month := 1, [1849].time.Day := 16, [1849].time.Hour := 2, [1849].time.Minute := 29, [1849].time.Second := 59, [1850].log_data[0].min := 1.0, [1850].log_data[0].max := 1.0, [1850].log_data[0].total := 300.0, [1850].log_data[0].time := 300.0, [1850].log_data[0].minminute := 30, [1850].log_data[0].maxminute := 30, [1850].log_data[0].valid := 1, [1850].log_data[1].valid := 1, [1850].log_data[2].valid := 1, [1850].log_data[3].valid := 1, [1850].log_data[4].valid := 1, [1850].log_data[5].valid := 1, [1850].log_data[6].valid := 1, [1850].log_data[7].valid := 1, [1850].log_data[8].valid := 1, [1850].log_data[9].valid := 1, [1850].log_data[10].valid := 1, [1850].log_data[11].valid := 1, [1850].log_data[12].valid := 1, [1850].log_data[13].valid := 1, [1850].log_data[14].valid := 1, [1850].log_data[15].valid := 1, [1850].log_data[16].valid := 1, [1850].log_data[17].valid := 1, [1850].log_data[18].valid := 1, [1850].log_data[19].valid := 1, [1850].time.Year := 2023, [1850].time.Month := 1, [1850].time.Day := 16, [1850].time.Hour := 2, [1850].time.Minute := 34, [1850].time.Second := 59, [1851].log_data[0].min := 1.0, [1851].log_data[0].max := 1.0, [1851].log_data[0].total := 300.0, [1851].log_data[0].time := 300.0, [1851].log_data[0].minminute := 35, [1851].log_data[0].maxminute := 35, [1851].log_data[0].valid := 1, [1851].log_data[1].valid := 1, [1851].log_data[2].valid := 1, [1851].log_data[3].valid := 1, [1851].log_data[4].valid := 1, [1851].log_data[5].valid := 1, [1851].log_data[6].valid := 1, [1851].log_data[7].valid := 1, [1851].log_data[8].valid := 1, [1851].log_data[9].valid := 1, [1851].log_data[10].valid := 1, [1851].log_data[11].valid := 1, [1851].log_data[12].valid := 1, [1851].log_data[13].valid := 1, [1851].log_data[14].valid := 1, [1851].log_data[15].valid := 1,
        [1851].log_data[16].valid := 1, [1851].log_data[17].valid := 1, [1851].log_data[18].valid := 1, [1851].log_data[19].valid := 1, [1851].time.Year := 2023, [1851].time.Month := 1, [1851].time.Day := 16, [1851].time.Hour := 2, [1851].time.Minute := 39, [1851].time.Second := 59, [1852].log_data[0].min := 1.0, [1852].log_data[0].max := 1.0, [1852].log_data[0].total := 300.0, [1852].log_data[0].time := 300.0, [1852].log_data[0].minminute := 40, [1852].log_data[0].maxminute := 40, [1852].log_data[0].valid := 1, [1852].log_data[1].valid := 1, [1852].log_data[2].valid := 1, [1852].log_data[3].valid := 1, [1852].log_data[4].valid := 1, [1852].log_data[5].valid := 1, [1852].log_data[6].valid := 1, [1852].log_data[7].valid := 1, [1852].log_data[8].valid := 1, [1852].log_data[9].valid := 1, [1852].log_data[10].valid := 1, [1852].log_data[11].valid := 1, [1852].log_data[12].valid := 1, [1852].log_data[13].valid := 1, [1852].log_data[14].valid := 1, [1852].log_data[15].valid := 1, [1852].log_data[16].valid := 1, [1852].log_data[17].valid := 1, [1852].log_data[18].valid := 1, [1852].log_data[19].valid := 1, [1852].time.Year := 2023, [1852].time.Month := 1, [1852].time.Day := 16, [1852].time.Hour := 2, [1852].time.Minute := 44, [1852].time.Second := 59, [1853].log_data[0].min := 1.0, [1853].log_data[0].max := 1.0, [1853].log_data[0].total := 300.0, [1853].log_data[0].time := 300.0, [1853].log_data[0].minminute := 45, [1853].log_data[0].maxminute := 45, [1853].log_data[0].valid := 1, [1853].log_data[1].valid := 1, [1853].log_data[2].valid := 1, [1853].log_data[3].valid := 1, [1853].log_data[4].valid := 1, [1853].log_data[5].valid := 1, [1853].log_data[6].valid := 1, [1853].log_data[7].valid := 1, [1853].log_data[8].valid := 1, [1853].log_data[9].valid := 1, [1853].log_data[10].valid := 1, [1853].log_data[11].valid := 1,
        [1853].log_data[12].valid := 1, [1853].log_data[13].valid := 1, [1853].log_data[14].valid := 1, [1853].log_data[15].valid := 1, [1853].log_data[16].valid := 1, [1853].log_data[17].valid := 1, [1853].log_data[18].valid := 1, [1853].log_data[19].valid := 1, [1853].time.Year := 2023, [1853].time.Month := 1, [1853].time.Day := 16, [1853].time.Hour := 2, [1853].time.Minute := 49, [1853].time.Second := 59, [1854].log_data[0].min := 1.0, [1854].log_data[0].max := 1.0, [1854].log_data[0].total := 300.0, [1854].log_data[0].time := 300.0, [1854].log_data[0].minminute := 50, [1854].log_data[0].maxminute := 50, [1854].log_data[0].valid := 1, [1854].log_data[1].valid := 1, [1854].log_data[2].valid := 1, [1854].log_data[3].valid := 1, [1854].log_data[4].valid := 1, [1854].log_data[5].valid := 1, [1854].log_data[6].valid := 1, [1854].log_data[7].valid := 1, [1854].log_data[8].valid := 1, [1854].log_data[9].valid := 1, [1854].log_data[10].valid := 1, [1854].log_data[11].valid := 1, [1854].log_data[12].valid := 1, [1854].log_data[13].valid := 1, [1854].log_data[14].valid := 1, [1854].log_data[15].valid := 1, [1854].log_data[16].valid := 1, [1854].log_data[17].valid := 1, [1854].log_data[18].valid := 1, [1854].log_data[19].valid := 1, [1854].time.Year := 2023, [1854].time.Month := 1, [1854].time.Day := 16, [1854].time.Hour := 2, [1854].time.Minute := 54, [1854].time.Second := 59, [1855].log_data[0].min := 1.0, [1855].log_data[0].max := 1.0, [1855].log_data[0].total := 300.0, [1855].log_data[0].time := 300.0, [1855].log_data[0].minminute := 55, [1855].log_data[0].maxminute := 55, [1855].log_data[0].valid := 1, [1855].log_data[1].valid := 1, [1855].log_data[2].valid := 1, [1855].log_data[3].valid := 1, [1855].log_data[4].valid := 1, [1855].log_data[5].valid := 1, [1855].log_data[6].valid := 1, [1855].log_data[7].valid := 1,
        [1855].log_data[8].valid := 1, [1855].log_data[9].valid := 1, [1855].log_data[10].valid := 1, [1855].log_data[11].valid := 1, [1855].log_data[12].valid := 1, [1855].log_data[13].valid := 1, [1855].log_data[14].valid := 1, [1855].log_data[15].valid := 1, [1855].log_data[16].valid := 1, [1855].log_data[17].valid := 1, [1855].log_data[18].valid := 1, [1855].log_data[19].valid := 1, [1855].time.Year := 2023, [1855].time.Month := 1, [1855].time.Day := 16, [1855].time.Hour := 2, [1855].time.Minute := 59, [1855].time.Second := 59, [1856].log_data[0].min := 1.0, [1856].log_data[0].max := 1.0, [1856].log_data[0].total := 300.0, [1856].log_data[0].time := 300.0, [1856].log_data[0].valid := 1, [1856].log_data[1].valid := 1, [1856].log_data[2].valid := 1, [1856].log_data[3].valid := 1, [1856].log_data[4].valid := 1, [1856].log_data[5].valid := 1, [1856].log_data[6].valid := 1, [1856].log_data[7].valid := 1, [1856].log_data[8].valid := 1, [1856].log_data[9].valid := 1, [1856].log_data[10].valid := 1, [1856].log_data[11].valid := 1, [1856].log_data[12].valid := 1, [1856].log_data[13].valid := 1, [1856].log_data[14].valid := 1, [1856].log_data[15].valid := 1, [1856].log_data[16].valid := 1, [1856].log_data[17].valid := 1, [1856].log_data[18].valid := 1, [1856].log_data[19].valid := 1, [1856].time.Year := 2023, [1856].time.Month := 1, [1856].time.Day := 16, [1856].time.Hour := 3, [1856].time.Minute := 4, [1856].time.Second := 59, [1857].log_data[0].min := 1.0, [1857].log_data[0].max := 1.0, [1857].log_data[0].total := 300.0, [1857].log_data[0].time := 300.0, [1857].log_data[0].minminute := 5, [1857].log_data[0].maxminute := 5, [1857].log_data[0].valid := 1, [1857].log_data[1].valid := 1, [1857].log_data[2].valid := 1, [1857].log_data[3].valid := 1, [1857].log_data[4].valid := 1, [1857].log_data[5].valid := 1,
        [1857].log_data[6].valid := 1, [1857].log_data[7].valid := 1, [1857].log_data[8].valid := 1, [1857].log_data[9].valid := 1, [1857].log_data[10].valid := 1, [1857].log_data[11].valid := 1, [1857].log_data[12].valid := 1, [1857].log_data[13].valid := 1, [1857].log_data[14].valid := 1, [1857].log_data[15].valid := 1, [1857].log_data[16].valid := 1, [1857].log_data[17].valid := 1, [1857].log_data[18].valid := 1, [1857].log_data[19].valid := 1, [1857].time.Year := 2023, [1857].time.Month := 1, [1857].time.Day := 16, [1857].time.Hour := 3, [1857].time.Minute := 9, [1857].time.Second := 59, [1858].log_data[0].min := 1.0, [1858].log_data[0].max := 1.0, [1858].log_data[0].total := 300.0, [1858].log_data[0].time := 300.0, [1858].log_data[0].minminute := 10, [1858].log_data[0].maxminute := 10, [1858].log_data[0].valid := 1, [1858].log_data[1].valid := 1, [1858].log_data[2].valid := 1, [1858].log_data[3].valid := 1, [1858].log_data[4].valid := 1, [1858].log_data[5].valid := 1, [1858].log_data[6].valid := 1, [1858].log_data[7].valid := 1, [1858].log_data[8].valid := 1, [1858].log_data[9].valid := 1, [1858].log_data[10].valid := 1, [1858].log_data[11].valid := 1, [1858].log_data[12].valid := 1, [1858].log_data[13].valid := 1, [1858].log_data[14].valid := 1, [1858].log_data[15].valid := 1, [1858].log_data[16].valid := 1, [1858].log_data[17].valid := 1, [1858].log_data[18].valid := 1, [1858].log_data[19].valid := 1, [1858].time.Year := 2023, [1858].time.Month := 1, [1858].time.Day := 16, [1858].time.Hour := 3, [1858].time.Minute := 14, [1858].time.Second := 59, [1859].log_data[0].min := 1.0, [1859].log_data[0].max := 1.0, [1859].log_data[0].total := 300.0, [1859].log_data[0].time := 300.0, [1859].log_data[0].minminute := 15, [1859].log_data[0].maxminute := 15, [1859].log_data[0].valid := 1, [1859].log_data[1].valid := 1,
        [1859].log_data[2].valid := 1, [1859].log_data[3].valid := 1, [1859].log_data[4].valid := 1, [1859].log_data[5].valid := 1, [1859].log_data[6].valid := 1, [1859].log_data[7].valid := 1, [1859].log_data[8].valid := 1, [1859].log_data[9].valid := 1, [1859].log_data[10].valid := 1, [1859].log_data[11].valid := 1, [1859].log_data[12].valid := 1, [1859].log_data[13].valid := 1, [1859].log_data[14].valid := 1, [1859].log_data[15].valid := 1, [1859].log_data[16].valid := 1, [1859].log_data[17].valid := 1, [1859].log_data[18].valid := 1, [1859].log_data[19].valid := 1, [1859].time.Year := 2023, [1859].time.Month := 1, [1859].time.Day := 16, [1859].time.Hour := 3, [1859].time.Minute := 19, [1859].time.Second := 59, [1860].log_data[0].min := 1.0, [1860].log_data[0].max := 1.0, [1860].log_data[0].total := 300.0, [1860].log_data[0].time := 300.0, [1860].log_data[0].minminute := 20, [1860].log_data[0].maxminute := 20, [1860].log_data[0].valid := 1, [1860].log_data[1].valid := 1, [1860].log_data[2].valid := 1, [1860].log_data[3].valid := 1, [1860].log_data[4].valid := 1, [1860].log_data[5].valid := 1, [1860].log_data[6].valid := 1, [1860].log_data[7].valid := 1, [1860].log_data[8].valid := 1, [1860].log_data[9].valid := 1, [1860].log_data[10].valid := 1, [1860].log_data[11].valid := 1, [1860].log_data[12].valid := 1, [1860].log_data[13].valid := 1, [1860].log_data[14].valid := 1, [1860].log_data[15].valid := 1, [1860].log_data[16].valid := 1, [1860].log_data[17].valid := 1, [1860].log_data[18].valid := 1, [1860].log_data[19].valid := 1, [1860].time.Year := 2023, [1860].time.Month := 1, [1860].time.Day := 16, [1860].time.Hour := 3, [1860].time.Minute := 24, [1860].time.Second := 59, [1861].log_data[0].min := 1.0, [1861].log_data[0].max := 1.0, [1861].log_data[0].total := 300.0, [1861].log_data[0].time := 300.0,
        [1861].log_data[0].minminute := 25, [1861].log_data[0].maxminute := 25, [1861].log_data[0].valid := 1, [1861].log_data[1].valid := 1, [1861].log_data[2].valid := 1, [1861].log_data[3].valid := 1, [1861].log_data[4].valid := 1, [1861].log_data[5].valid := 1, [1861].log_data[6].valid := 1, [1861].log_data[7].valid := 1, [1861].log_data[8].valid := 1, [1861].log_data[9].valid := 1, [1861].log_data[10].valid := 1, [1861].log_data[11].valid := 1, [1861].log_data[12].valid := 1, [1861].log_data[13].valid := 1, [1861].log_data[14].valid := 1, [1861].log_data[15].valid := 1, [1861].log_data[16].valid := 1, [1861].log_data[17].valid := 1, [1861].log_data[18].valid := 1, [1861].log_data[19].valid := 1, [1861].time.Year := 2023, [1861].time.Month := 1, [1861].time.Day := 16, [1861].time.Hour := 3, [1861].time.Minute := 29, [1861].time.Second := 59, [1862].log_data[0].min := 1.0, [1862].log_data[0].max := 1.0, [1862].log_data[0].total := 300.0, [1862].log_data[0].time := 300.0, [1862].log_data[0].minminute := 30, [1862].log_data[0].maxminute := 30, [1862].log_data[0].valid := 1, [1862].log_data[1].valid := 1, [1862].log_data[2].valid := 1, [1862].log_data[3].valid := 1, [1862].log_data[4].valid := 1, [1862].log_data[5].valid := 1, [1862].log_data[6].valid := 1, [1862].log_data[7].valid := 1, [1862].log_data[8].valid := 1, [1862].log_data[9].valid := 1, [1862].log_data[10].valid := 1, [1862].log_data[11].valid := 1, [1862].log_data[12].valid := 1, [1862].log_data[13].valid := 1, [1862].log_data[14].valid := 1, [1862].log_data[15].valid := 1, [1862].log_data[16].valid := 1, [1862].log_data[17].valid := 1, [1862].log_data[18].valid := 1, [1862].log_data[19].valid := 1, [1862].time.Year := 2023, [1862].time.Month := 1, [1862].time.Day := 16, [1862].time.Hour := 3, [1862].time.Minute := 34, [1862].time.Second := 59,
        [1863].log_data[0].min := 1.0, [1863].log_data[0].max := 1.0, [1863].log_data[0].total := 300.0, [1863].log_data[0].time := 300.0, [1863].log_data[0].minminute := 35, [1863].log_data[0].maxminute := 35, [1863].log_data[0].valid := 1, [1863].log_data[1].valid := 1, [1863].log_data[2].valid := 1, [1863].log_data[3].valid := 1, [1863].log_data[4].valid := 1, [1863].log_data[5].valid := 1, [1863].log_data[6].valid := 1, [1863].log_data[7].valid := 1, [1863].log_data[8].valid := 1, [1863].log_data[9].valid := 1, [1863].log_data[10].valid := 1, [1863].log_data[11].valid := 1, [1863].log_data[12].valid := 1, [1863].log_data[13].valid := 1, [1863].log_data[14].valid := 1, [1863].log_data[15].valid := 1, [1863].log_data[16].valid := 1, [1863].log_data[17].valid := 1, [1863].log_data[18].valid := 1, [1863].log_data[19].valid := 1, [1863].time.Year := 2023, [1863].time.Month := 1, [1863].time.Day := 16, [1863].time.Hour := 3, [1863].time.Minute := 39, [1863].time.Second := 59, [1864].log_data[0].min := 1.0, [1864].log_data[0].max := 1.0, [1864].log_data[0].total := 300.0, [1864].log_data[0].time := 300.0, [1864].log_data[0].minminute := 40, [1864].log_data[0].maxminute := 40, [1864].log_data[0].valid := 1, [1864].log_data[1].valid := 1, [1864].log_data[2].valid := 1, [1864].log_data[3].valid := 1, [1864].log_data[4].valid := 1, [1864].log_data[5].valid := 1, [1864].log_data[6].valid := 1, [1864].log_data[7].valid := 1, [1864].log_data[8].valid := 1, [1864].log_data[9].valid := 1, [1864].log_data[10].valid := 1, [1864].log_data[11].valid := 1, [1864].log_data[12].valid := 1, [1864].log_data[13].valid := 1, [1864].log_data[14].valid := 1, [1864].log_data[15].valid := 1, [1864].log_data[16].valid := 1, [1864].log_data[17].valid := 1, [1864].log_data[18].valid := 1, [1864].log_data[19].valid := 1, [1864].time.Year := 2023, [1864].time.Month := 1,
        [1864].time.Day := 16, [1864].time.Hour := 3, [1864].time.Minute := 44, [1864].time.Second := 59, [1865].log_data[0].min := 1.0, [1865].log_data[0].max := 1.0, [1865].log_data[0].total := 300.0, [1865].log_data[0].time := 300.0, [1865].log_data[0].minminute := 45, [1865].log_data[0].maxminute := 45, [1865].log_data[0].valid := 1, [1865].log_data[1].valid := 1, [1865].log_data[2].valid := 1, [1865].log_data[3].valid := 1, [1865].log_data[4].valid := 1, [1865].log_data[5].valid := 1, [1865].log_data[6].valid := 1, [1865].log_data[7].valid := 1, [1865].log_data[8].valid := 1, [1865].log_data[9].valid := 1, [1865].log_data[10].valid := 1, [1865].log_data[11].valid := 1, [1865].log_data[12].valid := 1, [1865].log_data[13].valid := 1, [1865].log_data[14].valid := 1, [1865].log_data[15].valid := 1, [1865].log_data[16].valid := 1, [1865].log_data[17].valid := 1, [1865].log_data[18].valid := 1, [1865].log_data[19].valid := 1, [1865].time.Year := 2023, [1865].time.Month := 1, [1865].time.Day := 16, [1865].time.Hour := 3, [1865].time.Minute := 49, [1865].time.Second := 59, [1866].log_data[0].min := 1.0, [1866].log_data[0].max := 1.0, [1866].log_data[0].total := 300.0, [1866].log_data[0].time := 300.0, [1866].log_data[0].minminute := 50, [1866].log_data[0].maxminute := 50, [1866].log_data[0].valid := 1, [1866].log_data[1].valid := 1, [1866].log_data[2].valid := 1, [1866].log_data[3].valid := 1, [1866].log_data[4].valid := 1, [1866].log_data[5].valid := 1, [1866].log_data[6].valid := 1, [1866].log_data[7].valid := 1, [1866].log_data[8].valid := 1, [1866].log_data[9].valid := 1, [1866].log_data[10].valid := 1, [1866].log_data[11].valid := 1, [1866].log_data[12].valid := 1, [1866].log_data[13].valid := 1, [1866].log_data[14].valid := 1, [1866].log_data[15].valid := 1, [1866].log_data[16].valid := 1, [1866].log_data[17].valid := 1,
        [1866].log_data[18].valid := 1, [1866].log_data[19].valid := 1, [1866].time.Year := 2023, [1866].time.Month := 1, [1866].time.Day := 16, [1866].time.Hour := 3, [1866].time.Minute := 54, [1866].time.Second := 59, [1867].log_data[0].min := 1.0, [1867].log_data[0].max := 1.0, [1867].log_data[0].total := 300.0, [1867].log_data[0].time := 300.0, [1867].log_data[0].minminute := 55, [1867].log_data[0].maxminute := 55, [1867].log_data[0].valid := 1, [1867].log_data[1].valid := 1, [1867].log_data[2].valid := 1, [1867].log_data[3].valid := 1, [1867].log_data[4].valid := 1, [1867].log_data[5].valid := 1, [1867].log_data[6].valid := 1, [1867].log_data[7].valid := 1, [1867].log_data[8].valid := 1, [1867].log_data[9].valid := 1, [1867].log_data[10].valid := 1, [1867].log_data[11].valid := 1, [1867].log_data[12].valid := 1, [1867].log_data[13].valid := 1, [1867].log_data[14].valid := 1, [1867].log_data[15].valid := 1, [1867].log_data[16].valid := 1, [1867].log_data[17].valid := 1, [1867].log_data[18].valid := 1, [1867].log_data[19].valid := 1, [1867].time.Year := 2023, [1867].time.Month := 1, [1867].time.Day := 16, [1867].time.Hour := 3, [1867].time.Minute := 59, [1867].time.Second := 59, [1868].log_data[0].min := 1.0, [1868].log_data[0].max := 1.0, [1868].log_data[0].total := 300.0, [1868].log_data[0].time := 300.0, [1868].log_data[0].valid := 1, [1868].log_data[1].valid := 1, [1868].log_data[2].valid := 1, [1868].log_data[3].valid := 1, [1868].log_data[4].valid := 1, [1868].log_data[5].valid := 1, [1868].log_data[6].valid := 1, [1868].log_data[7].valid := 1, [1868].log_data[8].valid := 1, [1868].log_data[9].valid := 1, [1868].log_data[10].valid := 1, [1868].log_data[11].valid := 1, [1868].log_data[12].valid := 1, [1868].log_data[13].valid := 1, [1868].log_data[14].valid := 1, [1868].log_data[15].valid := 1,
        [1868].log_data[16].valid := 1, [1868].log_data[17].valid := 1, [1868].log_data[18].valid := 1, [1868].log_data[19].valid := 1, [1868].time.Year := 2023, [1868].time.Month := 1, [1868].time.Day := 16, [1868].time.Hour := 4, [1868].time.Minute := 4, [1868].time.Second := 59, [1869].log_data[0].min := 1.0, [1869].log_data[0].max := 1.0, [1869].log_data[0].total := 300.0, [1869].log_data[0].time := 300.0, [1869].log_data[0].minminute := 5, [1869].log_data[0].maxminute := 5, [1869].log_data[0].valid := 1, [1869].log_data[1].valid := 1, [1869].log_data[2].valid := 1, [1869].log_data[3].valid := 1, [1869].log_data[4].valid := 1, [1869].log_data[5].valid := 1, [1869].log_data[6].valid := 1, [1869].log_data[7].valid := 1, [1869].log_data[8].valid := 1, [1869].log_data[9].valid := 1, [1869].log_data[10].valid := 1, [1869].log_data[11].valid := 1, [1869].log_data[12].valid := 1, [1869].log_data[13].valid := 1, [1869].log_data[14].valid := 1, [1869].log_data[15].valid := 1, [1869].log_data[16].valid := 1, [1869].log_data[17].valid := 1, [1869].log_data[18].valid := 1, [1869].log_data[19].valid := 1, [1869].time.Year := 2023, [1869].time.Month := 1, [1869].time.Day := 16, [1869].time.Hour := 4, [1869].time.Minute := 9, [1869].time.Second := 59, [1870].log_data[0].min := 1.0, [1870].log_data[0].max := 1.0, [1870].log_data[0].total := 300.0, [1870].log_data[0].time := 300.0, [1870].log_data[0].minminute := 10, [1870].log_data[0].maxminute := 10, [1870].log_data[0].valid := 1, [1870].log_data[1].valid := 1, [1870].log_data[2].valid := 1, [1870].log_data[3].valid := 1, [1870].log_data[4].valid := 1, [1870].log_data[5].valid := 1, [1870].log_data[6].valid := 1, [1870].log_data[7].valid := 1, [1870].log_data[8].valid := 1, [1870].log_data[9].valid := 1, [1870].log_data[10].valid := 1, [1870].log_data[11].valid := 1,
        [1870].log_data[12].valid := 1, [1870].log_data[13].valid := 1, [1870].log_data[14].valid := 1, [1870].log_data[15].valid := 1, [1870].log_data[16].valid := 1, [1870].log_data[17].valid := 1, [1870].log_data[18].valid := 1, [1870].log_data[19].valid := 1, [1870].time.Year := 2023, [1870].time.Month := 1, [1870].time.Day := 16, [1870].time.Hour := 4, [1870].time.Minute := 14, [1870].time.Second := 59, [1871].log_data[0].min := 1.0, [1871].log_data[0].max := 1.0, [1871].log_data[0].total := 300.0, [1871].log_data[0].time := 300.0, [1871].log_data[0].minminute := 15, [1871].log_data[0].maxminute := 15, [1871].log_data[0].valid := 1, [1871].log_data[1].valid := 1, [1871].log_data[2].valid := 1, [1871].log_data[3].valid := 1, [1871].log_data[4].valid := 1, [1871].log_data[5].valid := 1, [1871].log_data[6].valid := 1, [1871].log_data[7].valid := 1, [1871].log_data[8].valid := 1, [1871].log_data[9].valid := 1, [1871].log_data[10].valid := 1, [1871].log_data[11].valid := 1, [1871].log_data[12].valid := 1, [1871].log_data[13].valid := 1, [1871].log_data[14].valid := 1, [1871].log_data[15].valid := 1, [1871].log_data[16].valid := 1, [1871].log_data[17].valid := 1, [1871].log_data[18].valid := 1, [1871].log_data[19].valid := 1, [1871].time.Year := 2023, [1871].time.Month := 1, [1871].time.Day := 16, [1871].time.Hour := 4, [1871].time.Minute := 19, [1871].time.Second := 59, [1872].log_data[0].min := 1.0, [1872].log_data[0].max := 1.0, [1872].log_data[0].total := 300.0, [1872].log_data[0].time := 300.0, [1872].log_data[0].minminute := 20, [1872].log_data[0].maxminute := 20, [1872].log_data[0].valid := 1, [1872].log_data[1].valid := 1, [1872].log_data[2].valid := 1, [1872].log_data[3].valid := 1, [1872].log_data[4].valid := 1, [1872].log_data[5].valid := 1, [1872].log_data[6].valid := 1, [1872].log_data[7].valid := 1,
        [1872].log_data[8].valid := 1, [1872].log_data[9].valid := 1, [1872].log_data[10].valid := 1, [1872].log_data[11].valid := 1, [1872].log_data[12].valid := 1, [1872].log_data[13].valid := 1, [1872].log_data[14].valid := 1, [1872].log_data[15].valid := 1, [1872].log_data[16].valid := 1, [1872].log_data[17].valid := 1, [1872].log_data[18].valid := 1, [1872].log_data[19].valid := 1, [1872].time.Year := 2023, [1872].time.Month := 1, [1872].time.Day := 16, [1872].time.Hour := 4, [1872].time.Minute := 24, [1872].time.Second := 59, [1873].log_data[0].min := 1.0, [1873].log_data[0].max := 1.0, [1873].log_data[0].total := 300.0, [1873].log_data[0].time := 300.0, [1873].log_data[0].minminute := 25, [1873].log_data[0].maxminute := 25, [1873].log_data[0].valid := 1, [1873].log_data[1].valid := 1, [1873].log_data[2].valid := 1, [1873].log_data[3].valid := 1, [1873].log_data[4].valid := 1, [1873].log_data[5].valid := 1, [1873].log_data[6].valid := 1, [1873].log_data[7].valid := 1, [1873].log_data[8].valid := 1, [1873].log_data[9].valid := 1, [1873].log_data[10].valid := 1, [1873].log_data[11].valid := 1, [1873].log_data[12].valid := 1, [1873].log_data[13].valid := 1, [1873].log_data[14].valid := 1, [1873].log_data[15].valid := 1, [1873].log_data[16].valid := 1, [1873].log_data[17].valid := 1, [1873].log_data[18].valid := 1, [1873].log_data[19].valid := 1, [1873].time.Year := 2023, [1873].time.Month := 1, [1873].time.Day := 16, [1873].time.Hour := 4, [1873].time.Minute := 29, [1873].time.Second := 59, [1874].log_data[0].min := 1.0, [1874].log_data[0].max := 1.0, [1874].log_data[0].total := 300.0, [1874].log_data[0].time := 300.0, [1874].log_data[0].minminute := 30, [1874].log_data[0].maxminute := 30, [1874].log_data[0].valid := 1, [1874].log_data[1].valid := 1, [1874].log_data[2].valid := 1, [1874].log_data[3].valid := 1,
        [1874].log_data[4].valid := 1, [1874].log_data[5].valid := 1, [1874].log_data[6].valid := 1, [1874].log_data[7].valid := 1, [1874].log_data[8].valid := 1, [1874].log_data[9].valid := 1, [1874].log_data[10].valid := 1, [1874].log_data[11].valid := 1, [1874].log_data[12].valid := 1, [1874].log_data[13].valid := 1, [1874].log_data[14].valid := 1, [1874].log_data[15].valid := 1, [1874].log_data[16].valid := 1, [1874].log_data[17].valid := 1, [1874].log_data[18].valid := 1, [1874].log_data[19].valid := 1, [1874].time.Year := 2023, [1874].time.Month := 1, [1874].time.Day := 16, [1874].time.Hour := 4, [1874].time.Minute := 34, [1874].time.Second := 59, [1875].log_data[0].min := 1.0, [1875].log_data[0].max := 1.0, [1875].log_data[0].total := 300.0, [1875].log_data[0].time := 300.0, [1875].log_data[0].minminute := 35, [1875].log_data[0].maxminute := 35, [1875].log_data[0].valid := 1, [1875].log_data[1].valid := 1, [1875].log_data[2].valid := 1, [1875].log_data[3].valid := 1, [1875].log_data[4].valid := 1, [1875].log_data[5].valid := 1, [1875].log_data[6].valid := 1, [1875].log_data[7].valid := 1, [1875].log_data[8].valid := 1, [1875].log_data[9].valid := 1, [1875].log_data[10].valid := 1, [1875].log_data[11].valid := 1, [1875].log_data[12].valid := 1, [1875].log_data[13].valid := 1, [1875].log_data[14].valid := 1, [1875].log_data[15].valid := 1, [1875].log_data[16].valid := 1, [1875].log_data[17].valid := 1, [1875].log_data[18].valid := 1, [1875].log_data[19].valid := 1, [1875].time.Year := 2023, [1875].time.Month := 1, [1875].time.Day := 16, [1875].time.Hour := 4, [1875].time.Minute := 39, [1875].time.Second := 59, [1876].log_data[0].min := 1.0, [1876].log_data[0].max := 1.0, [1876].log_data[0].total := 300.0, [1876].log_data[0].time := 300.0, [1876].log_data[0].minminute := 40, [1876].log_data[0].maxminute := 40,
        [1876].log_data[0].valid := 1, [1876].log_data[1].valid := 1, [1876].log_data[2].valid := 1, [1876].log_data[3].valid := 1, [1876].log_data[4].valid := 1, [1876].log_data[5].valid := 1, [1876].log_data[6].valid := 1, [1876].log_data[7].valid := 1, [1876].log_data[8].valid := 1, [1876].log_data[9].valid := 1, [1876].log_data[10].valid := 1, [1876].log_data[11].valid := 1, [1876].log_data[12].valid := 1, [1876].log_data[13].valid := 1, [1876].log_data[14].valid := 1, [1876].log_data[15].valid := 1, [1876].log_data[16].valid := 1, [1876].log_data[17].valid := 1, [1876].log_data[18].valid := 1, [1876].log_data[19].valid := 1, [1876].time.Year := 2023, [1876].time.Month := 1, [1876].time.Day := 16, [1876].time.Hour := 4, [1876].time.Minute := 44, [1876].time.Second := 59, [1877].log_data[0].min := 1.0, [1877].log_data[0].max := 1.0, [1877].log_data[0].total := 300.0, [1877].log_data[0].time := 300.0, [1877].log_data[0].minminute := 45, [1877].log_data[0].maxminute := 45, [1877].log_data[0].valid := 1, [1877].log_data[1].valid := 1, [1877].log_data[2].valid := 1, [1877].log_data[3].valid := 1, [1877].log_data[4].valid := 1, [1877].log_data[5].valid := 1, [1877].log_data[6].valid := 1, [1877].log_data[7].valid := 1, [1877].log_data[8].valid := 1, [1877].log_data[9].valid := 1, [1877].log_data[10].valid := 1, [1877].log_data[11].valid := 1, [1877].log_data[12].valid := 1, [1877].log_data[13].valid := 1, [1877].log_data[14].valid := 1, [1877].log_data[15].valid := 1, [1877].log_data[16].valid := 1, [1877].log_data[17].valid := 1, [1877].log_data[18].valid := 1, [1877].log_data[19].valid := 1, [1877].time.Year := 2023, [1877].time.Month := 1, [1877].time.Day := 16, [1877].time.Hour := 4, [1877].time.Minute := 49, [1877].time.Second := 59, [1878].log_data[0].min := 1.0, [1878].log_data[0].max := 1.0,
        [1878].log_data[0].total := 300.0, [1878].log_data[0].time := 300.0, [1878].log_data[0].minminute := 50, [1878].log_data[0].maxminute := 50, [1878].log_data[0].valid := 1, [1878].log_data[1].valid := 1, [1878].log_data[2].valid := 1, [1878].log_data[3].valid := 1, [1878].log_data[4].valid := 1, [1878].log_data[5].valid := 1, [1878].log_data[6].valid := 1, [1878].log_data[7].valid := 1, [1878].log_data[8].valid := 1, [1878].log_data[9].valid := 1, [1878].log_data[10].valid := 1, [1878].log_data[11].valid := 1, [1878].log_data[12].valid := 1, [1878].log_data[13].valid := 1, [1878].log_data[14].valid := 1, [1878].log_data[15].valid := 1, [1878].log_data[16].valid := 1, [1878].log_data[17].valid := 1, [1878].log_data[18].valid := 1, [1878].log_data[19].valid := 1, [1878].time.Year := 2023, [1878].time.Month := 1, [1878].time.Day := 16, [1878].time.Hour := 4, [1878].time.Minute := 54, [1878].time.Second := 59, [1879].log_data[0].min := 1.0, [1879].log_data[0].max := 1.0, [1879].log_data[0].total := 300.0, [1879].log_data[0].time := 300.0, [1879].log_data[0].minminute := 55, [1879].log_data[0].maxminute := 55, [1879].log_data[0].valid := 1, [1879].log_data[1].valid := 1, [1879].log_data[2].valid := 1, [1879].log_data[3].valid := 1, [1879].log_data[4].valid := 1, [1879].log_data[5].valid := 1, [1879].log_data[6].valid := 1, [1879].log_data[7].valid := 1, [1879].log_data[8].valid := 1, [1879].log_data[9].valid := 1, [1879].log_data[10].valid := 1, [1879].log_data[11].valid := 1, [1879].log_data[12].valid := 1, [1879].log_data[13].valid := 1, [1879].log_data[14].valid := 1, [1879].log_data[15].valid := 1, [1879].log_data[16].valid := 1, [1879].log_data[17].valid := 1, [1879].log_data[18].valid := 1, [1879].log_data[19].valid := 1, [1879].time.Year := 2023, [1879].time.Month := 1, [1879].time.Day := 16, [1879].time.Hour := 4,
        [1879].time.Minute := 59, [1879].time.Second := 59, [1880].log_data[0].min := 1.0, [1880].log_data[0].max := 1.0, [1880].log_data[0].total := 300.0, [1880].log_data[0].time := 300.0, [1880].log_data[0].valid := 1, [1880].log_data[1].valid := 1, [1880].log_data[2].valid := 1, [1880].log_data[3].valid := 1, [1880].log_data[4].valid := 1, [1880].log_data[5].valid := 1, [1880].log_data[6].valid := 1, [1880].log_data[7].valid := 1, [1880].log_data[8].valid := 1, [1880].log_data[9].valid := 1, [1880].log_data[10].valid := 1, [1880].log_data[11].valid := 1, [1880].log_data[12].valid := 1, [1880].log_data[13].valid := 1, [1880].log_data[14].valid := 1, [1880].log_data[15].valid := 1, [1880].log_data[16].valid := 1, [1880].log_data[17].valid := 1, [1880].log_data[18].valid := 1, [1880].log_data[19].valid := 1, [1880].time.Year := 2023, [1880].time.Month := 1, [1880].time.Day := 16, [1880].time.Hour := 5, [1880].time.Minute := 4, [1880].time.Second := 59, [1881].log_data[0].min := 1.0, [1881].log_data[0].max := 1.0, [1881].log_data[0].total := 300.0, [1881].log_data[0].time := 300.0, [1881].log_data[0].minminute := 5, [1881].log_data[0].maxminute := 5, [1881].log_data[0].valid := 1, [1881].log_data[1].valid := 1, [1881].log_data[2].valid := 1, [1881].log_data[3].valid := 1, [1881].log_data[4].valid := 1, [1881].log_data[5].valid := 1, [1881].log_data[6].valid := 1, [1881].log_data[7].valid := 1, [1881].log_data[8].valid := 1, [1881].log_data[9].valid := 1, [1881].log_data[10].valid := 1, [1881].log_data[11].valid := 1, [1881].log_data[12].valid := 1, [1881].log_data[13].valid := 1, [1881].log_data[14].valid := 1, [1881].log_data[15].valid := 1, [1881].log_data[16].valid := 1, [1881].log_data[17].valid := 1, [1881].log_data[18].valid := 1, [1881].log_data[19].valid := 1, [1881].time.Year := 2023, [1881].time.Month := 1,
        [1881].time.Day := 16, [1881].time.Hour := 5, [1881].time.Minute := 9, [1881].time.Second := 59, [1882].log_data[0].min := 1.0, [1882].log_data[0].max := 1.0, [1882].log_data[0].total := 300.0, [1882].log_data[0].time := 300.0, [1882].log_data[0].minminute := 10, [1882].log_data[0].maxminute := 10, [1882].log_data[0].valid := 1, [1882].log_data[1].valid := 1, [1882].log_data[2].valid := 1, [1882].log_data[3].valid := 1, [1882].log_data[4].valid := 1, [1882].log_data[5].valid := 1, [1882].log_data[6].valid := 1, [1882].log_data[7].valid := 1, [1882].log_data[8].valid := 1, [1882].log_data[9].valid := 1, [1882].log_data[10].valid := 1, [1882].log_data[11].valid := 1, [1882].log_data[12].valid := 1, [1882].log_data[13].valid := 1, [1882].log_data[14].valid := 1, [1882].log_data[15].valid := 1, [1882].log_data[16].valid := 1, [1882].log_data[17].valid := 1, [1882].log_data[18].valid := 1, [1882].log_data[19].valid := 1, [1882].time.Year := 2023, [1882].time.Month := 1, [1882].time.Day := 16, [1882].time.Hour := 5, [1882].time.Minute := 14, [1882].time.Second := 59, [1883].log_data[0].min := 1.0, [1883].log_data[0].max := 1.0, [1883].log_data[0].total := 300.0, [1883].log_data[0].time := 300.0, [1883].log_data[0].minminute := 15, [1883].log_data[0].maxminute := 15, [1883].log_data[0].valid := 1, [1883].log_data[1].valid := 1, [1883].log_data[2].valid := 1, [1883].log_data[3].valid := 1, [1883].log_data[4].valid := 1, [1883].log_data[5].valid := 1, [1883].log_data[6].valid := 1, [1883].log_data[7].valid := 1, [1883].log_data[8].valid := 1, [1883].log_data[9].valid := 1, [1883].log_data[10].valid := 1, [1883].log_data[11].valid := 1, [1883].log_data[12].valid := 1, [1883].log_data[13].valid := 1, [1883].log_data[14].valid := 1, [1883].log_data[15].valid := 1, [1883].log_data[16].valid := 1, [1883].log_data[17].valid := 1,
        [1883].log_data[18].valid := 1, [1883].log_data[19].valid := 1, [1883].time.Year := 2023, [1883].time.Month := 1, [1883].time.Day := 16, [1883].time.Hour := 5, [1883].time.Minute := 19, [1883].time.Second := 59, [1884].log_data[0].min := 1.0, [1884].log_data[0].max := 1.0, [1884].log_data[0].total := 300.0, [1884].log_data[0].time := 300.0, [1884].log_data[0].minminute := 20, [1884].log_data[0].maxminute := 20, [1884].log_data[0].valid := 1, [1884].log_data[1].valid := 1, [1884].log_data[2].valid := 1, [1884].log_data[3].valid := 1, [1884].log_data[4].valid := 1, [1884].log_data[5].valid := 1, [1884].log_data[6].valid := 1, [1884].log_data[7].valid := 1, [1884].log_data[8].valid := 1, [1884].log_data[9].valid := 1, [1884].log_data[10].valid := 1, [1884].log_data[11].valid := 1, [1884].log_data[12].valid := 1, [1884].log_data[13].valid := 1, [1884].log_data[14].valid := 1, [1884].log_data[15].valid := 1, [1884].log_data[16].valid := 1, [1884].log_data[17].valid := 1, [1884].log_data[18].valid := 1, [1884].log_data[19].valid := 1, [1884].time.Year := 2023, [1884].time.Month := 1, [1884].time.Day := 16, [1884].time.Hour := 5, [1884].time.Minute := 24, [1884].time.Second := 59, [1885].log_data[0].min := 1.0, [1885].log_data[0].max := 1.0, [1885].log_data[0].total := 300.0, [1885].log_data[0].time := 300.0, [1885].log_data[0].minminute := 25, [1885].log_data[0].maxminute := 25, [1885].log_data[0].valid := 1, [1885].log_data[1].valid := 1, [1885].log_data[2].valid := 1, [1885].log_data[3].valid := 1, [1885].log_data[4].valid := 1, [1885].log_data[5].valid := 1, [1885].log_data[6].valid := 1, [1885].log_data[7].valid := 1, [1885].log_data[8].valid := 1, [1885].log_data[9].valid := 1, [1885].log_data[10].valid := 1, [1885].log_data[11].valid := 1, [1885].log_data[12].valid := 1, [1885].log_data[13].valid := 1,
        [1885].log_data[14].valid := 1, [1885].log_data[15].valid := 1, [1885].log_data[16].valid := 1, [1885].log_data[17].valid := 1, [1885].log_data[18].valid := 1, [1885].log_data[19].valid := 1, [1885].time.Year := 2023, [1885].time.Month := 1, [1885].time.Day := 16, [1885].time.Hour := 5, [1885].time.Minute := 29, [1885].time.Second := 59, [1886].log_data[0].min := 1.0, [1886].log_data[0].max := 1.0, [1886].log_data[0].total := 300.0, [1886].log_data[0].time := 300.0, [1886].log_data[0].minminute := 30, [1886].log_data[0].maxminute := 30, [1886].log_data[0].valid := 1, [1886].log_data[1].valid := 1, [1886].log_data[2].valid := 1, [1886].log_data[3].valid := 1, [1886].log_data[4].valid := 1, [1886].log_data[5].valid := 1, [1886].log_data[6].valid := 1, [1886].log_data[7].valid := 1, [1886].log_data[8].valid := 1, [1886].log_data[9].valid := 1, [1886].log_data[10].valid := 1, [1886].log_data[11].valid := 1, [1886].log_data[12].valid := 1, [1886].log_data[13].valid := 1, [1886].log_data[14].valid := 1, [1886].log_data[15].valid := 1, [1886].log_data[16].valid := 1, [1886].log_data[17].valid := 1, [1886].log_data[18].valid := 1, [1886].log_data[19].valid := 1, [1886].time.Year := 2023, [1886].time.Month := 1, [1886].time.Day := 16, [1886].time.Hour := 5, [1886].time.Minute := 34, [1886].time.Second := 59, [1887].log_data[0].min := 1.0, [1887].log_data[0].max := 1.0, [1887].log_data[0].total := 300.0, [1887].log_data[0].time := 300.0, [1887].log_data[0].minminute := 35, [1887].log_data[0].maxminute := 35, [1887].log_data[0].valid := 1, [1887].log_data[1].valid := 1, [1887].log_data[2].valid := 1, [1887].log_data[3].valid := 1, [1887].log_data[4].valid := 1, [1887].log_data[5].valid := 1, [1887].log_data[6].valid := 1, [1887].log_data[7].valid := 1, [1887].log_data[8].valid := 1, [1887].log_data[9].valid := 1,
        [1887].log_data[10].valid := 1, [1887].log_data[11].valid := 1, [1887].log_data[12].valid := 1, [1887].log_data[13].valid := 1, [1887].log_data[14].valid := 1, [1887].log_data[15].valid := 1, [1887].log_data[16].valid := 1, [1887].log_data[17].valid := 1, [1887].log_data[18].valid := 1, [1887].log_data[19].valid := 1, [1887].time.Year := 2023, [1887].time.Month := 1, [1887].time.Day := 16, [1887].time.Hour := 5, [1887].time.Minute := 39, [1887].time.Second := 59, [1888].log_data[0].min := 1.0, [1888].log_data[0].max := 1.0, [1888].log_data[0].total := 300.0, [1888].log_data[0].time := 300.0, [1888].log_data[0].minminute := 40, [1888].log_data[0].maxminute := 40, [1888].log_data[0].valid := 1, [1888].log_data[1].valid := 1, [1888].log_data[2].valid := 1, [1888].log_data[3].valid := 1, [1888].log_data[4].valid := 1, [1888].log_data[5].valid := 1, [1888].log_data[6].valid := 1, [1888].log_data[7].valid := 1, [1888].log_data[8].valid := 1, [1888].log_data[9].valid := 1, [1888].log_data[10].valid := 1, [1888].log_data[11].valid := 1, [1888].log_data[12].valid := 1, [1888].log_data[13].valid := 1, [1888].log_data[14].valid := 1, [1888].log_data[15].valid := 1, [1888].log_data[16].valid := 1, [1888].log_data[17].valid := 1, [1888].log_data[18].valid := 1, [1888].log_data[19].valid := 1, [1888].time.Year := 2023, [1888].time.Month := 1, [1888].time.Day := 16, [1888].time.Hour := 5, [1888].time.Minute := 44, [1888].time.Second := 59, [1889].log_data[0].min := 1.0, [1889].log_data[0].max := 1.0, [1889].log_data[0].total := 300.0, [1889].log_data[0].time := 300.0, [1889].log_data[0].minminute := 45, [1889].log_data[0].maxminute := 45, [1889].log_data[0].valid := 1, [1889].log_data[1].valid := 1, [1889].log_data[2].valid := 1, [1889].log_data[3].valid := 1, [1889].log_data[4].valid := 1, [1889].log_data[5].valid := 1,
        [1889].log_data[6].valid := 1, [1889].log_data[7].valid := 1, [1889].log_data[8].valid := 1, [1889].log_data[9].valid := 1, [1889].log_data[10].valid := 1, [1889].log_data[11].valid := 1, [1889].log_data[12].valid := 1, [1889].log_data[13].valid := 1, [1889].log_data[14].valid := 1, [1889].log_data[15].valid := 1, [1889].log_data[16].valid := 1, [1889].log_data[17].valid := 1, [1889].log_data[18].valid := 1, [1889].log_data[19].valid := 1, [1889].time.Year := 2023, [1889].time.Month := 1, [1889].time.Day := 16, [1889].time.Hour := 5, [1889].time.Minute := 49, [1889].time.Second := 59, [1890].log_data[0].min := 1.0, [1890].log_data[0].max := 1.0, [1890].log_data[0].total := 300.0, [1890].log_data[0].time := 300.0, [1890].log_data[0].minminute := 50, [1890].log_data[0].maxminute := 50, [1890].log_data[0].valid := 1, [1890].log_data[1].valid := 1, [1890].log_data[2].valid := 1, [1890].log_data[3].valid := 1, [1890].log_data[4].valid := 1, [1890].log_data[5].valid := 1, [1890].log_data[6].valid := 1, [1890].log_data[7].valid := 1, [1890].log_data[8].valid := 1, [1890].log_data[9].valid := 1, [1890].log_data[10].valid := 1, [1890].log_data[11].valid := 1, [1890].log_data[12].valid := 1, [1890].log_data[13].valid := 1, [1890].log_data[14].valid := 1, [1890].log_data[15].valid := 1, [1890].log_data[16].valid := 1, [1890].log_data[17].valid := 1, [1890].log_data[18].valid := 1, [1890].log_data[19].valid := 1, [1890].time.Year := 2023, [1890].time.Month := 1, [1890].time.Day := 16, [1890].time.Hour := 5, [1890].time.Minute := 54, [1890].time.Second := 59, [1891].log_data[0].min := 1.0, [1891].log_data[0].max := 1.0, [1891].log_data[0].total := 300.0, [1891].log_data[0].time := 300.0, [1891].log_data[0].minminute := 55, [1891].log_data[0].maxminute := 55, [1891].log_data[0].valid := 1, [1891].log_data[1].valid := 1,
        [1891].log_data[2].valid := 1, [1891].log_data[3].valid := 1, [1891].log_data[4].valid := 1, [1891].log_data[5].valid := 1, [1891].log_data[6].valid := 1, [1891].log_data[7].valid := 1, [1891].log_data[8].valid := 1, [1891].log_data[9].valid := 1, [1891].log_data[10].valid := 1, [1891].log_data[11].valid := 1, [1891].log_data[12].valid := 1, [1891].log_data[13].valid := 1, [1891].log_data[14].valid := 1, [1891].log_data[15].valid := 1, [1891].log_data[16].valid := 1, [1891].log_data[17].valid := 1, [1891].log_data[18].valid := 1, [1891].log_data[19].valid := 1, [1891].time.Year := 2023, [1891].time.Month := 1, [1891].time.Day := 16, [1891].time.Hour := 5, [1891].time.Minute := 59, [1891].time.Second := 59, [1892].log_data[0].min := 1.0, [1892].log_data[0].max := 1.0, [1892].log_data[0].total := 300.0, [1892].log_data[0].time := 300.0, [1892].log_data[0].valid := 1, [1892].log_data[1].valid := 1, [1892].log_data[2].valid := 1, [1892].log_data[3].valid := 1, [1892].log_data[4].valid := 1, [1892].log_data[5].valid := 1, [1892].log_data[6].valid := 1, [1892].log_data[7].valid := 1, [1892].log_data[8].valid := 1, [1892].log_data[9].valid := 1, [1892].log_data[10].valid := 1, [1892].log_data[11].valid := 1, [1892].log_data[12].valid := 1, [1892].log_data[13].valid := 1, [1892].log_data[14].valid := 1, [1892].log_data[15].valid := 1, [1892].log_data[16].valid := 1, [1892].log_data[17].valid := 1, [1892].log_data[18].valid := 1, [1892].log_data[19].valid := 1, [1892].time.Year := 2023, [1892].time.Month := 1, [1892].time.Day := 16, [1892].time.Hour := 6, [1892].time.Minute := 4, [1892].time.Second := 59, [1893].log_data[0].min := 1.0, [1893].log_data[0].max := 1.0, [1893].log_data[0].total := 300.0, [1893].log_data[0].time := 300.0, [1893].log_data[0].minminute := 5, [1893].log_data[0].maxminute := 5,
        [1893].log_data[0].valid := 1, [1893].log_data[1].valid := 1, [1893].log_data[2].valid := 1, [1893].log_data[3].valid := 1, [1893].log_data[4].valid := 1, [1893].log_data[5].valid := 1, [1893].log_data[6].valid := 1, [1893].log_data[7].valid := 1, [1893].log_data[8].valid := 1, [1893].log_data[9].valid := 1, [1893].log_data[10].valid := 1, [1893].log_data[11].valid := 1, [1893].log_data[12].valid := 1, [1893].log_data[13].valid := 1, [1893].log_data[14].valid := 1, [1893].log_data[15].valid := 1, [1893].log_data[16].valid := 1, [1893].log_data[17].valid := 1, [1893].log_data[18].valid := 1, [1893].log_data[19].valid := 1, [1893].time.Year := 2023, [1893].time.Month := 1, [1893].time.Day := 16, [1893].time.Hour := 6, [1893].time.Minute := 9, [1893].time.Second := 59, [1894].log_data[0].min := 1.0, [1894].log_data[0].max := 1.0, [1894].log_data[0].total := 300.0, [1894].log_data[0].time := 300.0, [1894].log_data[0].minminute := 10, [1894].log_data[0].maxminute := 10, [1894].log_data[0].valid := 1, [1894].log_data[1].valid := 1, [1894].log_data[2].valid := 1, [1894].log_data[3].valid := 1, [1894].log_data[4].valid := 1, [1894].log_data[5].valid := 1, [1894].log_data[6].valid := 1, [1894].log_data[7].valid := 1, [1894].log_data[8].valid := 1, [1894].log_data[9].valid := 1, [1894].log_data[10].valid := 1, [1894].log_data[11].valid := 1, [1894].log_data[12].valid := 1, [1894].log_data[13].valid := 1, [1894].log_data[14].valid := 1, [1894].log_data[15].valid := 1, [1894].log_data[16].valid := 1, [1894].log_data[17].valid := 1, [1894].log_data[18].valid := 1, [1894].log_data[19].valid := 1, [1894].time.Year := 2023, [1894].time.Month := 1, [1894].time.Day := 16, [1894].time.Hour := 6, [1894].time.Minute := 14, [1894].time.Second := 59, [1895].log_data[0].min := 1.0, [1895].log_data[0].max := 1.0,
        [1895].log_data[0].total := 300.0, [1895].log_data[0].time := 300.0, [1895].log_data[0].minminute := 15, [1895].log_data[0].maxminute := 15, [1895].log_data[0].valid := 1, [1895].log_data[1].valid := 1, [1895].log_data[2].valid := 1, [1895].log_data[3].valid := 1, [1895].log_data[4].valid := 1, [1895].log_data[5].valid := 1, [1895].log_data[6].valid := 1, [1895].log_data[7].valid := 1, [1895].log_data[8].valid := 1, [1895].log_data[9].valid := 1, [1895].log_data[10].valid := 1, [1895].log_data[11].valid := 1, [1895].log_data[12].valid := 1, [1895].log_data[13].valid := 1, [1895].log_data[14].valid := 1, [1895].log_data[15].valid := 1, [1895].log_data[16].valid := 1, [1895].log_data[17].valid := 1, [1895].log_data[18].valid := 1, [1895].log_data[19].valid := 1, [1895].time.Year := 2023, [1895].time.Month := 1, [1895].time.Day := 16, [1895].time.Hour := 6, [1895].time.Minute := 19, [1895].time.Second := 59, [1896].log_data[0].min := 1.0, [1896].log_data[0].max := 1.0, [1896].log_data[0].total := 300.0, [1896].log_data[0].time := 300.0, [1896].log_data[0].minminute := 20, [1896].log_data[0].maxminute := 20, [1896].log_data[0].valid := 1, [1896].log_data[1].valid := 1, [1896].log_data[2].valid := 1, [1896].log_data[3].valid := 1, [1896].log_data[4].valid := 1, [1896].log_data[5].valid := 1, [1896].log_data[6].valid := 1, [1896].log_data[7].valid := 1, [1896].log_data[8].valid := 1, [1896].log_data[9].valid := 1, [1896].log_data[10].valid := 1, [1896].log_data[11].valid := 1, [1896].log_data[12].valid := 1, [1896].log_data[13].valid := 1, [1896].log_data[14].valid := 1, [1896].log_data[15].valid := 1, [1896].log_data[16].valid := 1, [1896].log_data[17].valid := 1, [1896].log_data[18].valid := 1, [1896].log_data[19].valid := 1, [1896].time.Year := 2023, [1896].time.Month := 1, [1896].time.Day := 16, [1896].time.Hour := 6,
        [1896].time.Minute := 24, [1896].time.Second := 59, [1897].log_data[0].min := 1.0, [1897].log_data[0].max := 1.0, [1897].log_data[0].total := 300.0, [1897].log_data[0].time := 300.0, [1897].log_data[0].minminute := 25, [1897].log_data[0].maxminute := 25, [1897].log_data[0].valid := 1, [1897].log_data[1].valid := 1, [1897].log_data[2].valid := 1, [1897].log_data[3].valid := 1, [1897].log_data[4].valid := 1, [1897].log_data[5].valid := 1, [1897].log_data[6].valid := 1, [1897].log_data[7].valid := 1, [1897].log_data[8].valid := 1, [1897].log_data[9].valid := 1, [1897].log_data[10].valid := 1, [1897].log_data[11].valid := 1, [1897].log_data[12].valid := 1, [1897].log_data[13].valid := 1, [1897].log_data[14].valid := 1, [1897].log_data[15].valid := 1, [1897].log_data[16].valid := 1, [1897].log_data[17].valid := 1, [1897].log_data[18].valid := 1, [1897].log_data[19].valid := 1, [1897].time.Year := 2023, [1897].time.Month := 1, [1897].time.Day := 16, [1897].time.Hour := 6, [1897].time.Minute := 29, [1897].time.Second := 59, [1898].log_data[0].min := 1.0, [1898].log_data[0].max := 1.0, [1898].log_data[0].total := 300.0, [1898].log_data[0].time := 300.0, [1898].log_data[0].minminute := 30, [1898].log_data[0].maxminute := 30, [1898].log_data[0].valid := 1, [1898].log_data[1].valid := 1, [1898].log_data[2].valid := 1, [1898].log_data[3].valid := 1, [1898].log_data[4].valid := 1, [1898].log_data[5].valid := 1, [1898].log_data[6].valid := 1, [1898].log_data[7].valid := 1, [1898].log_data[8].valid := 1, [1898].log_data[9].valid := 1, [1898].log_data[10].valid := 1, [1898].log_data[11].valid := 1, [1898].log_data[12].valid := 1, [1898].log_data[13].valid := 1, [1898].log_data[14].valid := 1, [1898].log_data[15].valid := 1, [1898].log_data[16].valid := 1, [1898].log_data[17].valid := 1, [1898].log_data[18].valid := 1, [1898].log_data[19].valid := 1,
        [1898].time.Year := 2023, [1898].time.Month := 1, [1898].time.Day := 16, [1898].time.Hour := 6, [1898].time.Minute := 34, [1898].time.Second := 59, [1899].log_data[0].min := 1.0, [1899].log_data[0].max := 1.0, [1899].log_data[0].total := 300.0, [1899].log_data[0].time := 300.0, [1899].log_data[0].minminute := 35, [1899].log_data[0].maxminute := 35, [1899].log_data[0].valid := 1, [1899].log_data[1].valid := 1, [1899].log_data[2].valid := 1, [1899].log_data[3].valid := 1, [1899].log_data[4].valid := 1, [1899].log_data[5].valid := 1, [1899].log_data[6].valid := 1, [1899].log_data[7].valid := 1, [1899].log_data[8].valid := 1, [1899].log_data[9].valid := 1, [1899].log_data[10].valid := 1, [1899].log_data[11].valid := 1, [1899].log_data[12].valid := 1, [1899].log_data[13].valid := 1, [1899].log_data[14].valid := 1, [1899].log_data[15].valid := 1, [1899].log_data[16].valid := 1, [1899].log_data[17].valid := 1, [1899].log_data[18].valid := 1, [1899].log_data[19].valid := 1, [1899].time.Year := 2023, [1899].time.Month := 1, [1899].time.Day := 16, [1899].time.Hour := 6, [1899].time.Minute := 39, [1899].time.Second := 59, [1900].log_data[0].min := 1.0, [1900].log_data[0].max := 1.0, [1900].log_data[0].total := 300.0, [1900].log_data[0].time := 300.0, [1900].log_data[0].minminute := 40, [1900].log_data[0].maxminute := 40, [1900].log_data[0].valid := 1, [1900].log_data[1].valid := 1, [1900].log_data[2].valid := 1, [1900].log_data[3].valid := 1, [1900].log_data[4].valid := 1, [1900].log_data[5].valid := 1, [1900].log_data[6].valid := 1, [1900].log_data[7].valid := 1, [1900].log_data[8].valid := 1, [1900].log_data[9].valid := 1, [1900].log_data[10].valid := 1, [1900].log_data[11].valid := 1, [1900].log_data[12].valid := 1, [1900].log_data[13].valid := 1, [1900].log_data[14].valid := 1, [1900].log_data[15].valid := 1,
        [1900].log_data[16].valid := 1, [1900].log_data[17].valid := 1, [1900].log_data[18].valid := 1, [1900].log_data[19].valid := 1, [1900].time.Year := 2023, [1900].time.Month := 1, [1900].time.Day := 16, [1900].time.Hour := 6, [1900].time.Minute := 44, [1900].time.Second := 59, [1901].log_data[0].min := 1.0, [1901].log_data[0].max := 1.0, [1901].log_data[0].total := 300.0, [1901].log_data[0].time := 300.0, [1901].log_data[0].minminute := 45, [1901].log_data[0].maxminute := 45, [1901].log_data[0].valid := 1, [1901].log_data[1].valid := 1, [1901].log_data[2].valid := 1, [1901].log_data[3].valid := 1, [1901].log_data[4].valid := 1, [1901].log_data[5].valid := 1, [1901].log_data[6].valid := 1, [1901].log_data[7].valid := 1, [1901].log_data[8].valid := 1, [1901].log_data[9].valid := 1, [1901].log_data[10].valid := 1, [1901].log_data[11].valid := 1, [1901].log_data[12].valid := 1, [1901].log_data[13].valid := 1, [1901].log_data[14].valid := 1, [1901].log_data[15].valid := 1, [1901].log_data[16].valid := 1, [1901].log_data[17].valid := 1, [1901].log_data[18].valid := 1, [1901].log_data[19].valid := 1, [1901].time.Year := 2023, [1901].time.Month := 1, [1901].time.Day := 16, [1901].time.Hour := 6, [1901].time.Minute := 49, [1901].time.Second := 59, [1902].log_data[0].min := 1.0, [1902].log_data[0].max := 1.0, [1902].log_data[0].total := 300.0, [1902].log_data[0].time := 300.0, [1902].log_data[0].minminute := 50, [1902].log_data[0].maxminute := 50, [1902].log_data[0].valid := 1, [1902].log_data[1].valid := 1, [1902].log_data[2].valid := 1, [1902].log_data[3].valid := 1, [1902].log_data[4].valid := 1, [1902].log_data[5].valid := 1, [1902].log_data[6].valid := 1, [1902].log_data[7].valid := 1, [1902].log_data[8].valid := 1, [1902].log_data[9].valid := 1, [1902].log_data[10].valid := 1, [1902].log_data[11].valid := 1,
        [1902].log_data[12].valid := 1, [1902].log_data[13].valid := 1, [1902].log_data[14].valid := 1, [1902].log_data[15].valid := 1, [1902].log_data[16].valid := 1, [1902].log_data[17].valid := 1, [1902].log_data[18].valid := 1, [1902].log_data[19].valid := 1, [1902].time.Year := 2023, [1902].time.Month := 1, [1902].time.Day := 16, [1902].time.Hour := 6, [1902].time.Minute := 54, [1902].time.Second := 59, [1903].log_data[0].min := 1.0, [1903].log_data[0].max := 1.0, [1903].log_data[0].total := 300.0, [1903].log_data[0].time := 300.0, [1903].log_data[0].minminute := 55, [1903].log_data[0].maxminute := 55, [1903].log_data[0].valid := 1, [1903].log_data[1].valid := 1, [1903].log_data[2].valid := 1, [1903].log_data[3].valid := 1, [1903].log_data[4].valid := 1, [1903].log_data[5].valid := 1, [1903].log_data[6].valid := 1, [1903].log_data[7].valid := 1, [1903].log_data[8].valid := 1, [1903].log_data[9].valid := 1, [1903].log_data[10].valid := 1, [1903].log_data[11].valid := 1, [1903].log_data[12].valid := 1, [1903].log_data[13].valid := 1, [1903].log_data[14].valid := 1, [1903].log_data[15].valid := 1, [1903].log_data[16].valid := 1, [1903].log_data[17].valid := 1, [1903].log_data[18].valid := 1, [1903].log_data[19].valid := 1, [1903].time.Year := 2023, [1903].time.Month := 1, [1903].time.Day := 16, [1903].time.Hour := 6, [1903].time.Minute := 59, [1903].time.Second := 59, [1904].log_data[0].min := 1.0, [1904].log_data[0].max := 1.0, [1904].log_data[0].total := 300.0, [1904].log_data[0].time := 300.0, [1904].log_data[0].valid := 1, [1904].log_data[1].valid := 1, [1904].log_data[2].valid := 1, [1904].log_data[3].valid := 1, [1904].log_data[4].valid := 1, [1904].log_data[5].valid := 1, [1904].log_data[6].valid := 1, [1904].log_data[7].valid := 1, [1904].log_data[8].valid := 1, [1904].log_data[9].valid := 1,
        [1904].log_data[10].valid := 1, [1904].log_data[11].valid := 1, [1904].log_data[12].valid := 1, [1904].log_data[13].valid := 1, [1904].log_data[14].valid := 1, [1904].log_data[15].valid := 1, [1904].log_data[16].valid := 1, [1904].log_data[17].valid := 1, [1904].log_data[18].valid := 1, [1904].log_data[19].valid := 1, [1904].time.Year := 2023, [1904].time.Month := 1, [1904].time.Day := 16, [1904].time.Hour := 7, [1904].time.Minute := 4, [1904].time.Second := 59, [1905].log_data[0].min := 1.0, [1905].log_data[0].max := 1.0, [1905].log_data[0].total := 300.0, [1905].log_data[0].time := 300.0, [1905].log_data[0].minminute := 5, [1905].log_data[0].maxminute := 5, [1905].log_data[0].valid := 1, [1905].log_data[1].valid := 1, [1905].log_data[2].valid := 1, [1905].log_data[3].valid := 1, [1905].log_data[4].valid := 1, [1905].log_data[5].valid := 1, [1905].log_data[6].valid := 1, [1905].log_data[7].valid := 1, [1905].log_data[8].valid := 1, [1905].log_data[9].valid := 1, [1905].log_data[10].valid := 1, [1905].log_data[11].valid := 1, [1905].log_data[12].valid := 1, [1905].log_data[13].valid := 1, [1905].log_data[14].valid := 1, [1905].log_data[15].valid := 1, [1905].log_data[16].valid := 1, [1905].log_data[17].valid := 1, [1905].log_data[18].valid := 1, [1905].log_data[19].valid := 1, [1905].time.Year := 2023, [1905].time.Month := 1, [1905].time.Day := 16, [1905].time.Hour := 7, [1905].time.Minute := 9, [1905].time.Second := 59, [1906].log_data[0].min := 1.0, [1906].log_data[0].max := 1.0, [1906].log_data[0].total := 300.0, [1906].log_data[0].time := 300.0, [1906].log_data[0].minminute := 10, [1906].log_data[0].maxminute := 10, [1906].log_data[0].valid := 1, [1906].log_data[1].valid := 1, [1906].log_data[2].valid := 1, [1906].log_data[3].valid := 1, [1906].log_data[4].valid := 1, [1906].log_data[5].valid := 1,
        [1906].log_data[6].valid := 1, [1906].log_data[7].valid := 1, [1906].log_data[8].valid := 1, [1906].log_data[9].valid := 1, [1906].log_data[10].valid := 1, [1906].log_data[11].valid := 1, [1906].log_data[12].valid := 1, [1906].log_data[13].valid := 1, [1906].log_data[14].valid := 1, [1906].log_data[15].valid := 1, [1906].log_data[16].valid := 1, [1906].log_data[17].valid := 1, [1906].log_data[18].valid := 1, [1906].log_data[19].valid := 1, [1906].time.Year := 2023, [1906].time.Month := 1, [1906].time.Day := 16, [1906].time.Hour := 7, [1906].time.Minute := 14, [1906].time.Second := 59, [1907].log_data[0].min := 1.0, [1907].log_data[0].max := 1.0, [1907].log_data[0].total := 300.0, [1907].log_data[0].time := 300.0, [1907].log_data[0].minminute := 15, [1907].log_data[0].maxminute := 15, [1907].log_data[0].valid := 1, [1907].log_data[1].valid := 1, [1907].log_data[2].valid := 1, [1907].log_data[3].valid := 1, [1907].log_data[4].valid := 1, [1907].log_data[5].valid := 1, [1907].log_data[6].valid := 1, [1907].log_data[7].valid := 1, [1907].log_data[8].valid := 1, [1907].log_data[9].valid := 1, [1907].log_data[10].valid := 1, [1907].log_data[11].valid := 1, [1907].log_data[12].valid := 1, [1907].log_data[13].valid := 1, [1907].log_data[14].valid := 1, [1907].log_data[15].valid := 1, [1907].log_data[16].valid := 1, [1907].log_data[17].valid := 1, [1907].log_data[18].valid := 1, [1907].log_data[19].valid := 1, [1907].time.Year := 2023, [1907].time.Month := 1, [1907].time.Day := 16, [1907].time.Hour := 7, [1907].time.Minute := 19, [1907].time.Second := 59, [1908].log_data[0].min := 1.0, [1908].log_data[0].max := 1.0, [1908].log_data[0].total := 300.0, [1908].log_data[0].time := 300.0, [1908].log_data[0].minminute := 20, [1908].log_data[0].maxminute := 20, [1908].log_data[0].valid := 1, [1908].log_data[1].valid := 1,
        [1908].log_data[2].valid := 1, [1908].log_data[3].valid := 1, [1908].log_data[4].valid := 1, [1908].log_data[5].valid := 1, [1908].log_data[6].valid := 1, [1908].log_data[7].valid := 1, [1908].log_data[8].valid := 1, [1908].log_data[9].valid := 1, [1908].log_data[10].valid := 1, [1908].log_data[11].valid := 1, [1908].log_data[12].valid := 1, [1908].log_data[13].valid := 1, [1908].log_data[14].valid := 1, [1908].log_data[15].valid := 1, [1908].log_data[16].valid := 1, [1908].log_data[17].valid := 1, [1908].log_data[18].valid := 1, [1908].log_data[19].valid := 1, [1908].time.Year := 2023, [1908].time.Month := 1, [1908].time.Day := 16, [1908].time.Hour := 7, [1908].time.Minute := 24, [1908].time.Second := 59, [1909].log_data[0].min := 1.0, [1909].log_data[0].max := 1.0, [1909].log_data[0].total := 300.0, [1909].log_data[0].time := 300.0, [1909].log_data[0].minminute := 25, [1909].log_data[0].maxminute := 25, [1909].log_data[0].valid := 1, [1909].log_data[1].valid := 1, [1909].log_data[2].valid := 1, [1909].log_data[3].valid := 1, [1909].log_data[4].valid := 1, [1909].log_data[5].valid := 1, [1909].log_data[6].valid := 1, [1909].log_data[7].valid := 1, [1909].log_data[8].valid := 1, [1909].log_data[9].valid := 1, [1909].log_data[10].valid := 1, [1909].log_data[11].valid := 1, [1909].log_data[12].valid := 1, [1909].log_data[13].valid := 1, [1909].log_data[14].valid := 1, [1909].log_data[15].valid := 1, [1909].log_data[16].valid := 1, [1909].log_data[17].valid := 1, [1909].log_data[18].valid := 1, [1909].log_data[19].valid := 1, [1909].time.Year := 2023, [1909].time.Month := 1, [1909].time.Day := 16, [1909].time.Hour := 7, [1909].time.Minute := 29, [1909].time.Second := 59, [1910].log_data[0].min := 1.0, [1910].log_data[0].max := 1.0, [1910].log_data[0].total := 300.0, [1910].log_data[0].time := 300.0,
        [1910].log_data[0].minminute := 30, [1910].log_data[0].maxminute := 30, [1910].log_data[0].valid := 1, [1910].log_data[1].valid := 1, [1910].log_data[2].valid := 1, [1910].log_data[3].valid := 1, [1910].log_data[4].valid := 1, [1910].log_data[5].valid := 1, [1910].log_data[6].valid := 1, [1910].log_data[7].valid := 1, [1910].log_data[8].valid := 1, [1910].log_data[9].valid := 1, [1910].log_data[10].valid := 1, [1910].log_data[11].valid := 1, [1910].log_data[12].valid := 1, [1910].log_data[13].valid := 1, [1910].log_data[14].valid := 1, [1910].log_data[15].valid := 1, [1910].log_data[16].valid := 1, [1910].log_data[17].valid := 1, [1910].log_data[18].valid := 1, [1910].log_data[19].valid := 1, [1910].time.Year := 2023, [1910].time.Month := 1, [1910].time.Day := 16, [1910].time.Hour := 7, [1910].time.Minute := 34, [1910].time.Second := 59, [1911].log_data[0].min := 1.0, [1911].log_data[0].max := 1.0, [1911].log_data[0].total := 300.0, [1911].log_data[0].time := 300.0, [1911].log_data[0].minminute := 35, [1911].log_data[0].maxminute := 35, [1911].log_data[0].valid := 1, [1911].log_data[1].valid := 1, [1911].log_data[2].valid := 1, [1911].log_data[3].valid := 1, [1911].log_data[4].valid := 1, [1911].log_data[5].valid := 1, [1911].log_data[6].valid := 1, [1911].log_data[7].valid := 1, [1911].log_data[8].valid := 1, [1911].log_data[9].valid := 1, [1911].log_data[10].valid := 1, [1911].log_data[11].valid := 1, [1911].log_data[12].valid := 1, [1911].log_data[13].valid := 1, [1911].log_data[14].valid := 1, [1911].log_data[15].valid := 1, [1911].log_data[16].valid := 1, [1911].log_data[17].valid := 1, [1911].log_data[18].valid := 1, [1911].log_data[19].valid := 1, [1911].time.Year := 2023, [1911].time.Month := 1, [1911].time.Day := 16, [1911].time.Hour := 7, [1911].time.Minute := 39, [1911].time.Second := 59,
